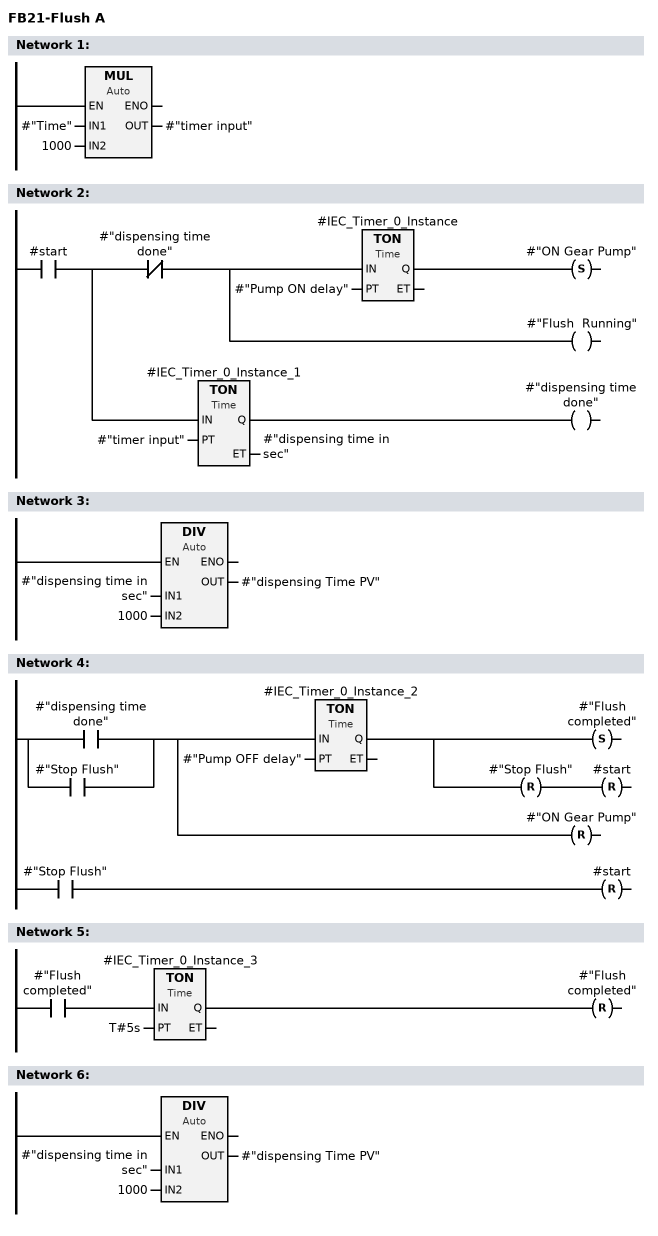
   RUNG wire#powerrail
      Mul(in1 := #"Time", in2 := 1000, out => #"timer input")
   END_RUNG
   // the same network as SCL:
   #"timer input" := #"Time" * 1000;
END_REGION

REGION Network 2
   RUNG wire#powerrail
      Contact( #start )
      wire#w1
      I_Contact( #"dispensing time done" )
      wire#w2
      { S7_Templates := "time_type := Time" } #IEC_Timer_0_Instance.TON(pt := #"Pump ON delay", et =>)
      S_Coil( #"ON Gear Pump" )
   END_RUNG
   RUNG wire#w2
      Coil( #"Flush  Running" )
   END_RUNG
   RUNG wire#w1
      { S7_Templates := "time_type := Time" } #IEC_Timer_0_Instance_1.TON(pt := #"timer input", et => #"dispensing time in sec")
      Coil( #"dispensing time done" )
   END_RUNG
   // the same network as SCL:
   #_w1 := #start AND NOT #"dispensing time done";
   #IEC_Timer_0_Instance(IN := #_w1, PT := #"Pump ON delay");   // TON
   IF #IEC_Timer_0_Instance.Q THEN #"ON Gear Pump" := TRUE; END_IF;
   #"Flush  Running" := #_w1;
   #IEC_Timer_0_Instance_1(IN := #start, PT := #"timer input", ET => #"dispensing time in sec");   // TON
   #"dispensing time done" := #IEC_Timer_0_Instance_1.Q;
END_REGION

REGION Network 3
   RUNG wire#powerrail
      Div(in1 := #"dispensing time in sec", in2 := 1000, out => #"dispensing Time PV")
   END_RUNG
   // the same network as SCL:
   #"dispensing Time PV" := #"dispensing time in sec" / 1000;
END_REGION

REGION Network 4
   RUNG wire#powerrail
      Contact( #"dispensing time done" )
      wire#w1
      { S7_Templates := "time_type := Time" } #IEC_Timer_0_Instance_2.TON(pt := #"Pump OFF delay", et =>)
      wire#w2
      S_Coil( #"Flush completed" )
   END_RUNG
   RUNG wire#powerrail
      Contact( #"Stop Flush" )
   END_RUNG wire#w1
   RUNG wire#w2
      R_Coil( #"Stop Flush" )
      R_Coil( #start )
   END_RUNG
   RUNG wire#w1
      R_Coil( #"ON Gear Pump" )
   END_RUNG
   RUNG wire#powerrail
      Contact( #"Stop Flush" )
      R_Coil( #start )
   END_RUNG
   // the same network as SCL:
   #_w1 := #"dispensing time done" OR #"Stop Flush";
   #IEC_Timer_0_Instance_2(IN := #_w1, PT := #"Pump OFF delay");   // TON
   IF #IEC_Timer_0_Instance_2.Q THEN
       #"Flush completed" := TRUE;
       #"Stop Flush" := FALSE;
       #start := FALSE;
   END_IF;
   IF #_w1 THEN #"ON Gear Pump" := FALSE; END_IF;
   IF #"Stop Flush" THEN #start := FALSE; END_IF;
END_REGION

REGION Network 5
   RUNG wire#powerrail
      Contact( #"Flush completed" )
      { S7_Templates := "time_type := Time" } #IEC_Timer_0_Instance_3.TON(pt := T#5s, et =>)
      R_Coil( #"Flush completed" )
   END_RUNG
   // the same network as SCL:
   #IEC_Timer_0_Instance_3(IN := #"Flush completed", PT := T#5s);   // TON
   IF #IEC_Timer_0_Instance_3.Q THEN #"Flush completed" := FALSE; END_IF;
END_REGION

REGION Network 6
   RUNG wire#powerrail
      Div(in1 := #"dispensing time in sec", in2 := 1000, out => #"dispensing Time PV")
   END_RUNG
   // the same network as SCL:
   #"dispensing Time PV" := #"dispensing time in sec" / 1000;
END_REGION
END_FUNCTION_BLOCK

FUNCTION "Regenaration program sequences" : Void   // FC23, LAD
{ S7_Optimized_Access := 'TRUE' }
VERSION : 0.1
// stored: AutoNumber true, IsIECCheckEnabled false, SetENOAutomatically false, UDAEnableTagReadback false
   VAR_TEMP
      temp1 : Bool;
   END_VAR
   VAR_TEMP   // added for the SCL form of the ladder/FBD networks
      _w1 : Bool;
   END_VAR
BEGIN

REGION Network 1: Function regeneration
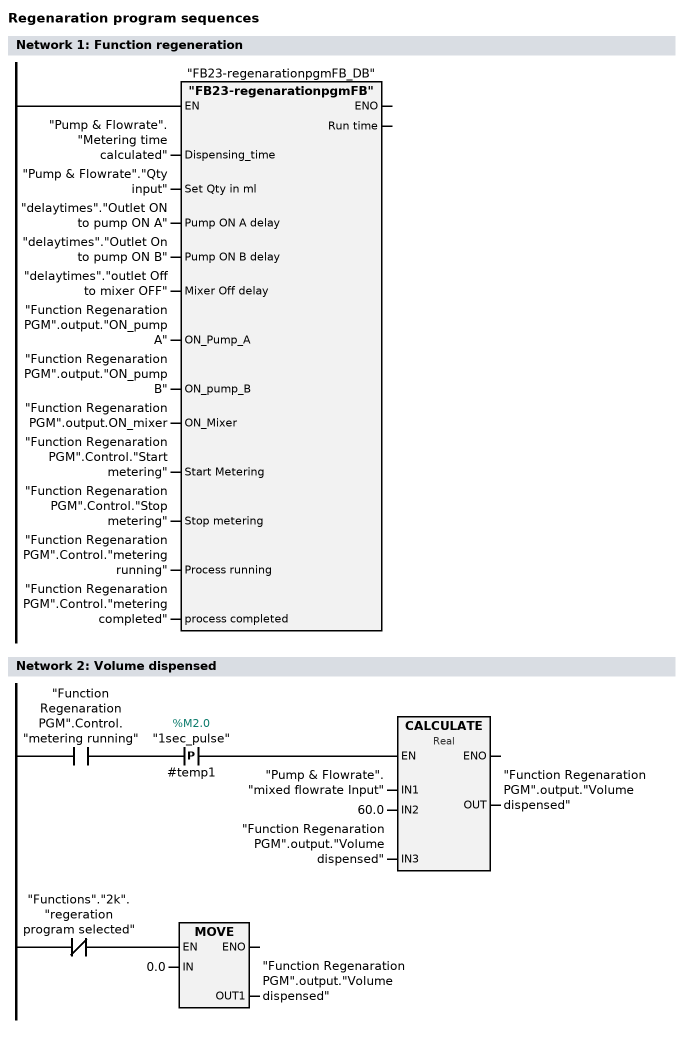
   RUNG wire#powerrail
      "FB23-regenarationpgmFB_DB"(Dispensing_time := "Pump & Flowrate"."Metering time calculated", "Set Qty in ml" := "Pump & Flowrate"."Qty input", "Pump ON A delay" := "delaytimes"."Outlet ON to pump ON A", "Pump ON B delay" := "delaytimes"."Outlet On to pump ON B", "Mixer Off delay" := "delaytimes"."outlet Off to mixer OFF", ON_Pump_A := "Function Regenaration PGM".output."ON_pump A", ON_pump_B := "Function Regenaration PGM".output."ON_pump B", ON_Mixer := "Function Regenaration PGM".output.ON_mixer, "Start Metering" := "Function Regenaration PGM".Control."Start metering", "Stop metering" := "Function Regenaration PGM".Control."Stop metering", "Process running" := "Function Regenaration PGM".Control."metering running", "process completed" := "Function Regenaration PGM".Control."metering completed", "Run time" =>)
   END_RUNG
   // the same network as SCL:
   "FB23-regenarationpgmFB_DB"(Dispensing_time := "Pump & Flowrate"."Metering time calculated",   // "FB23-regenarationpgmFB"
                           "Set Qty in ml" := "Pump & Flowrate"."Qty input",
                           "Pump ON A delay" := "delaytimes"."Outlet ON to pump ON A",
                           "Pump ON B delay" := "delaytimes"."Outlet On to pump ON B",
                           "Mixer Off delay" := "delaytimes"."outlet Off to mixer OFF",
                           ON_Pump_A := "Function Regenaration PGM".output."ON_pump A",
                           ON_pump_B := "Function Regenaration PGM".output."ON_pump B",
                           ON_Mixer := "Function Regenaration PGM".output.ON_mixer,
                           "Start Metering" := "Function Regenaration PGM".Control."Start metering",
                           "Stop metering" := "Function Regenaration PGM".Control."Stop metering",
                           "Process running" := "Function Regenaration PGM".Control."metering running",
                           "process completed" := "Function Regenaration PGM".Control."metering completed");
END_REGION

REGION Network 2: Volume dispensed
   RUNG wire#powerrail
      Contact( "Function Regenaration PGM".Control."metering running" )
      P_Contact(operand := "1sec_pulse", bit := #temp1)
      { S7_Templates := "SrcType := Real"; S7_Expression := "(IN1/IN2)+IN3" } Calculate(in1 := "Pump & Flowrate"."mixed flowrate Input", in2 := 60.0, in3 := "Function Regenaration PGM".output."Volume dispensed", out => "Function Regenaration PGM".output."Volume dispensed")
   END_RUNG
   RUNG wire#powerrail
      I_Contact( "Functions"."2k"."regeration program selected" )
      Move(in := 0.0, out1 => "Function Regenaration PGM".output."Volume dispensed")
   END_RUNG
   // the same network as SCL:
   #_w1 := "Function Regenaration PGM".Control."metering running" AND "1sec_pulse" AND NOT #temp1;   // rising edge of "1sec_pulse"
   #temp1 := "1sec_pulse";
   IF #_w1 THEN
       "Function Regenaration PGM".output."Volume dispensed" := ("Pump & Flowrate"."mixed flowrate Input"/60.0)+"Function Regenaration PGM".output."Volume dispensed";
   END_IF;
   IF NOT "Functions"."2k"."regeration program selected" THEN
       "Function Regenaration PGM".output."Volume dispensed" := 0.0;
   END_IF;
END_REGION
END_FUNCTION

FUNCTION_BLOCK "FB23-regenarationpgmFB"   // FB23, LAD
{ S7_Optimized_Access := 'TRUE' }
VERSION : 0.1
// stored: AutoNumber false, IsIECCheckEnabled false, IsRetainMemResEnabled false, MemoryReserve 100, SetENOAutomatically false, UDAEnableTagReadback false
   VAR_INPUT
      Dispensing_time : DInt;
      "Set Qty in ml" : Real;
      "Pump ON A delay" : DInt;
      "Pump ON B delay" : DInt;
      "Mixer Off delay" : DInt;
   END_VAR
   VAR_OUTPUT
      "Run time" : Int;
   END_VAR
   VAR_IN_OUT
      ON_Pump_A : Bool;
      ON_pump_B : Bool;
      ON_Mixer : Bool;
      "Start Metering" : Bool;
      "Stop metering" : Bool;
      "Process running" : Bool;
      "process completed" : Bool;
   END_VAR
   VAR
      "Total Volume dispensed" : Real;
      "metering started" : Bool;
      "metering time in msec" : DInt;
      "dispense time elapsed" : Bool;
   END_VAR
   VAR_TEMP
      Ons_temp : Bool;
   END_VAR
   VAR_TEMP   // added for the SCL form of the ladder/FBD networks
      _w1 : Bool;
   END_VAR
BEGIN

REGION Network 1
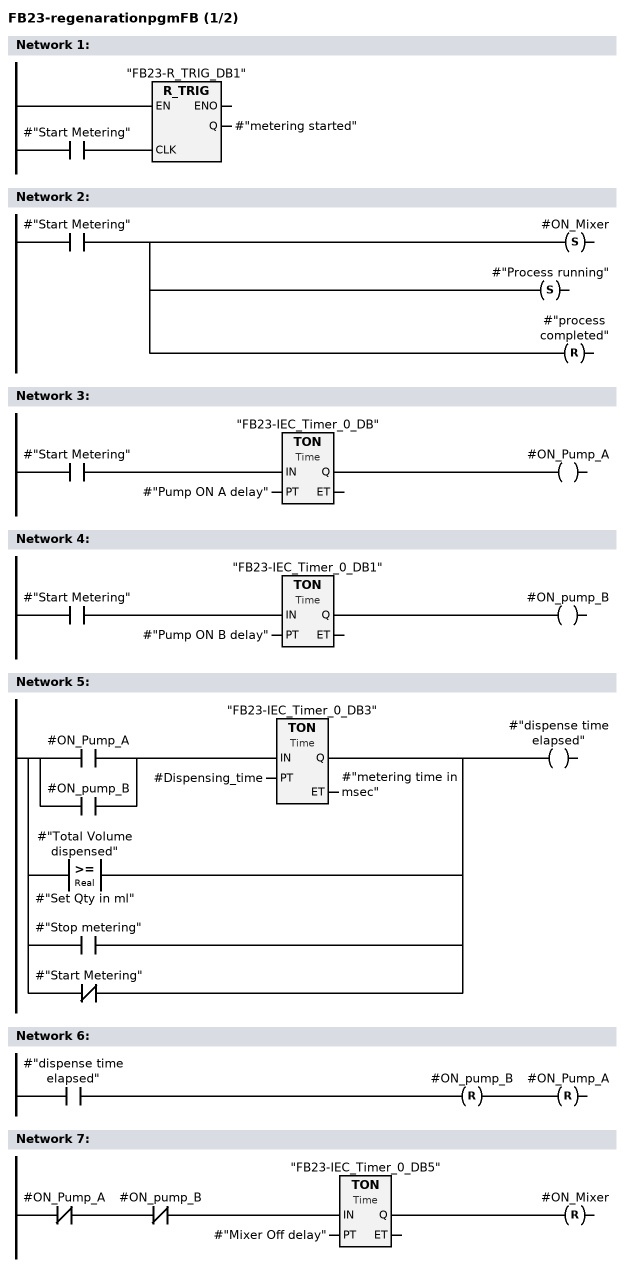
   RUNG wire#powerrail
      "FB23-R_TRIG_DB1".R_TRIG(CLK := wire#w1, Q => #"metering started")
   END_RUNG
   RUNG wire#powerrail
      Contact( #"Start Metering" )
   END_RUNG wire#w1
   // the same network as SCL:
   "FB23-R_TRIG_DB1"(CLK := #"Start Metering", Q => #"metering started");   // R_TRIG
END_REGION

REGION Network 2
   RUNG wire#powerrail
      Contact( #"Start Metering" )
      wire#w1
      S_Coil( #ON_Mixer )
   END_RUNG
   RUNG wire#w1
      S_Coil( #"Process running" )
   END_RUNG
   RUNG wire#w1
      R_Coil( #"process completed" )
   END_RUNG
   // the same network as SCL:
   IF #"Start Metering" THEN
       #ON_Mixer := TRUE;
       #"Process running" := TRUE;
       #"process completed" := FALSE;
   END_IF;
END_REGION

REGION Network 3
   RUNG wire#powerrail
      Contact( #"Start Metering" )
      { S7_Templates := "time_type := Time" } "FB23-IEC_Timer_0_DB".TON(pt := #"Pump ON A delay", et =>)
      Coil( #ON_Pump_A )
   END_RUNG
   // the same network as SCL:
   "FB23-IEC_Timer_0_DB".TON(IN := #"Start Metering", PT := #"Pump ON A delay");
   #ON_Pump_A := "FB23-IEC_Timer_0_DB".Q;
END_REGION

REGION Network 4
   RUNG wire#powerrail
      Contact( #"Start Metering" )
      { S7_Templates := "time_type := Time" } "FB23-IEC_Timer_0_DB1".TON(pt := #"Pump ON B delay", et =>)
      Coil( #ON_pump_B )
   END_RUNG
   // the same network as SCL:
   "FB23-IEC_Timer_0_DB1".TON(IN := #"Start Metering", PT := #"Pump ON B delay");
   #ON_pump_B := "FB23-IEC_Timer_0_DB1".Q;
END_REGION

REGION Network 5
   RUNG wire#powerrail
      Contact( #ON_Pump_A )
      wire#w1
      { S7_Templates := "time_type := Time" } "FB23-IEC_Timer_0_DB3".TON(pt := #Dispensing_time, et => #"metering time in msec")
      wire#w2
      Coil( #"dispense time elapsed" )
   END_RUNG
   RUNG wire#powerrail
      Contact( #ON_pump_B )
   END_RUNG wire#w1
   RUNG wire#powerrail
      { S7_Templates := "SrcType := Real" } GE_Contact(in1 := #"Total Volume dispensed", in2 := #"Set Qty in ml")
   END_RUNG wire#w2
   RUNG wire#powerrail
      Contact( #"Stop metering" )
   END_RUNG wire#w2
   RUNG wire#powerrail
      I_Contact( #"Start Metering" )
   END_RUNG wire#w2
   // the same network as SCL:
   "FB23-IEC_Timer_0_DB3".TON(IN := #ON_Pump_A OR #ON_pump_B,
                           PT := #Dispensing_time,
                           ET => #"metering time in msec");
   #"dispense time elapsed" := "FB23-IEC_Timer_0_DB3".Q OR (#"Total Volume dispensed" >= #"Set Qty in ml") OR #"Stop metering" OR NOT #"Start Metering";
END_REGION

REGION Network 6
   RUNG wire#powerrail
      Contact( #"dispense time elapsed" )
      R_Coil( #ON_pump_B )
      R_Coil( #ON_Pump_A )
   END_RUNG
   // the same network as SCL:
   IF #"dispense time elapsed" THEN
       #ON_pump_B := FALSE;
       #ON_Pump_A := FALSE;
   END_IF;
END_REGION

REGION Network 7
   RUNG wire#powerrail
      I_Contact( #ON_Pump_A )
      I_Contact( #ON_pump_B )
      { S7_Templates := "time_type := Time" } "FB23-IEC_Timer_0_DB5".TON(pt := #"Mixer Off delay", et =>)
      R_Coil( #ON_Mixer )
   END_RUNG
   // the same network as SCL:
   "FB23-IEC_Timer_0_DB5".TON(IN := NOT #ON_Pump_A AND NOT #ON_pump_B, PT := #"Mixer Off delay");
   IF "FB23-IEC_Timer_0_DB5".Q THEN #ON_Mixer := FALSE; END_IF;
END_REGION

REGION Network 8
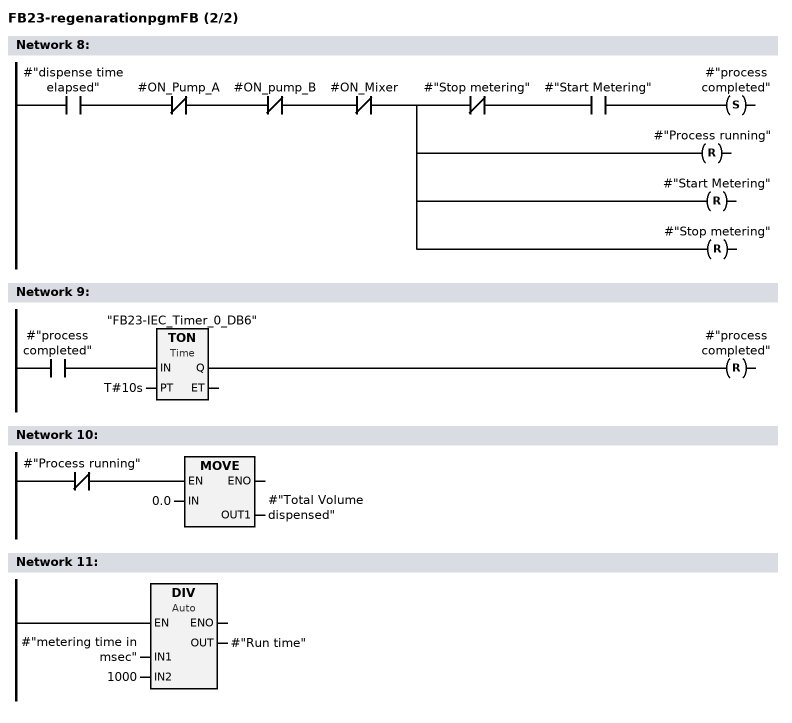
   RUNG wire#powerrail
      Contact( #"dispense time elapsed" )
      I_Contact( #ON_Pump_A )
      I_Contact( #ON_pump_B )
      I_Contact( #ON_Mixer )
      wire#w1
      I_Contact( #"Stop metering" )
      Contact( #"Start Metering" )
      S_Coil( #"process completed" )
   END_RUNG
   RUNG wire#w1
      R_Coil( #"Process running" )
   END_RUNG
   RUNG wire#w1
      R_Coil( #"Start Metering" )
   END_RUNG
   RUNG wire#w1
      R_Coil( #"Stop metering" )
   END_RUNG
   // the same network as SCL:
   #_w1 := #"dispense time elapsed" AND NOT #ON_Pump_A AND NOT #ON_pump_B AND NOT #ON_Mixer;
   IF #_w1 AND NOT #"Stop metering" AND #"Start Metering" THEN #"process completed" := TRUE; END_IF;
   IF #_w1 THEN
       #"Process running" := FALSE;
       #"Start Metering" := FALSE;
       #"Stop metering" := FALSE;
   END_IF;
END_REGION

REGION Network 9
   RUNG wire#powerrail
      Contact( #"process completed" )
      { S7_Templates := "time_type := Time" } "FB23-IEC_Timer_0_DB6".TON(pt := T#10s, et =>)
      R_Coil( #"process completed" )
   END_RUNG
   // the same network as SCL:
   "FB23-IEC_Timer_0_DB6".TON(IN := #"process completed", PT := T#10s);
   IF "FB23-IEC_Timer_0_DB6".Q THEN #"process completed" := FALSE; END_IF;
END_REGION

REGION Network 10
   RUNG wire#powerrail
      I_Contact( #"Process running" )
      Move(in := 0.0, out1 => #"Total Volume dispensed")
   END_RUNG
   // the same network as SCL:
   IF NOT #"Process running" THEN #"Total Volume dispensed" := 0.0; END_IF;
END_REGION

REGION Network 11
   RUNG wire#powerrail
      Div(in1 := #"metering time in msec", in2 := 1000, out => #"Run time")
   END_RUNG
   // the same network as SCL:
   #"Run time" := #"metering time in msec" / 1000;
END_REGION
END_FUNCTION_BLOCK

FUNCTION "Recirculation Sequences" : Void   // FC12, LAD
{ S7_Optimized_Access := 'TRUE' }
VERSION : 0.1
// stored: AutoNumber true, IsIECCheckEnabled false, SetENOAutomatically false, UDAEnableTagReadback false
   VAR_TEMP   // added for the SCL form of the ladder/FBD networks
      _w1 : Bool;
   END_VAR
BEGIN

REGION Network 1: A selection
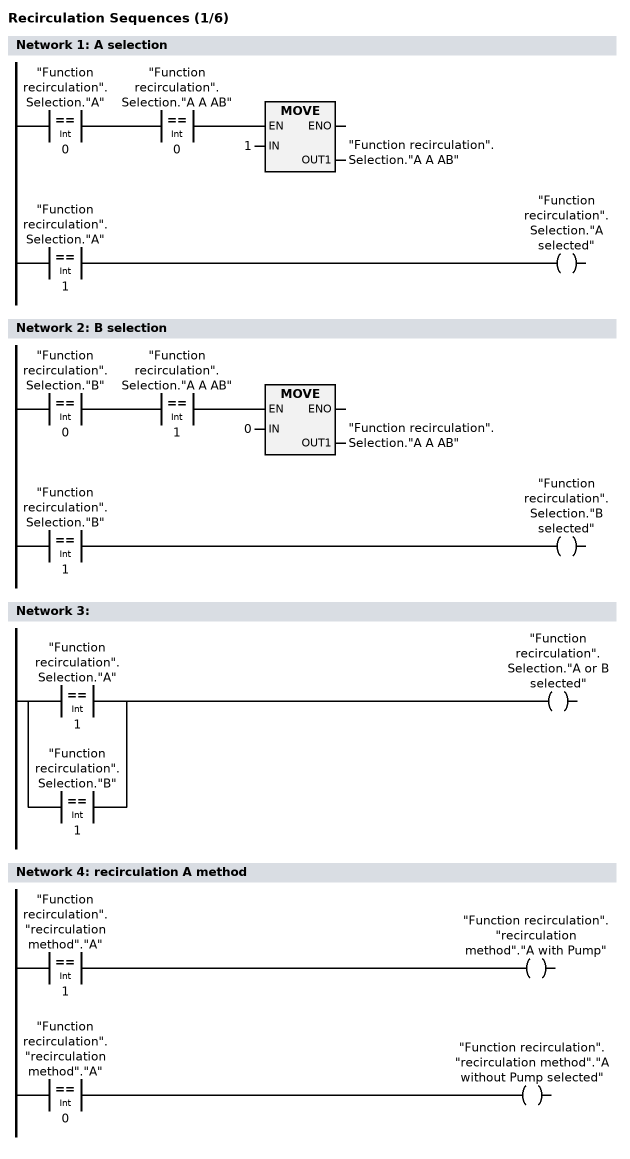
   RUNG wire#powerrail
      { S7_Templates := "SrcType := Int" } EQ_Contact(in1 := "Function recirculation".Selection."A", in2 := 0)
      { S7_Templates := "SrcType := Int" } EQ_Contact(in1 := "Function recirculation".Selection."A A AB", in2 := 0)
      Move(in := 1, out1 => "Function recirculation".Selection."A A AB")
   END_RUNG
   RUNG wire#powerrail
      { S7_Templates := "SrcType := Int" } EQ_Contact(in1 := "Function recirculation".Selection."A", in2 := 1)
      Coil( "Function recirculation".Selection."A selected" )
   END_RUNG
   // the same network as SCL:
   IF ("Function recirculation".Selection."A" = 0) AND ("Function recirculation".Selection."A A AB" = 0) THEN
       "Function recirculation".Selection."A A AB" := 1;
   END_IF;
   "Function recirculation".Selection."A selected" := "Function recirculation".Selection."A" = 1;
END_REGION

REGION Network 2: B selection
   RUNG wire#powerrail
      { S7_Templates := "SrcType := Int" } EQ_Contact(in1 := "Function recirculation".Selection."B", in2 := 0)
      { S7_Templates := "SrcType := Int" } EQ_Contact(in1 := "Function recirculation".Selection."A A AB", in2 := 1)
      Move(in := 0, out1 => "Function recirculation".Selection."A A AB")
   END_RUNG
   RUNG wire#powerrail
      { S7_Templates := "SrcType := Int" } EQ_Contact(in1 := "Function recirculation".Selection."B", in2 := 1)
      Coil( "Function recirculation".Selection."B selected" )
   END_RUNG
   // the same network as SCL:
   IF ("Function recirculation".Selection."B" = 0) AND ("Function recirculation".Selection."A A AB" = 1) THEN
       "Function recirculation".Selection."A A AB" := 0;
   END_IF;
   "Function recirculation".Selection."B selected" := "Function recirculation".Selection."B" = 1;
END_REGION

REGION Network 3
   RUNG wire#powerrail
      { S7_Templates := "SrcType := Int" } EQ_Contact(in1 := "Function recirculation".Selection."A", in2 := 1)
      wire#w1
      Coil( "Function recirculation".Selection."A or B selected" )
   END_RUNG
   RUNG wire#powerrail
      { S7_Templates := "SrcType := Int" } EQ_Contact(in1 := "Function recirculation".Selection."B", in2 := 1)
   END_RUNG wire#w1
   // the same network as SCL:
   "Function recirculation".Selection."A or B selected" := ("Function recirculation".Selection."A" = 1) OR ("Function recirculation".Selection."B" = 1);
END_REGION

REGION Network 4: recirculation A method
   RUNG wire#powerrail
      { S7_Templates := "SrcType := Int" } EQ_Contact(in1 := "Function recirculation"."recirculation method"."A", in2 := 1)
      Coil( "Function recirculation"."recirculation method"."A with Pump" )
   END_RUNG
   RUNG wire#powerrail
      { S7_Templates := "SrcType := Int" } EQ_Contact(in1 := "Function recirculation"."recirculation method"."A", in2 := 0)
      Coil( "Function recirculation"."recirculation method"."A without Pump selected" )
   END_RUNG
   // the same network as SCL:
   "Function recirculation"."recirculation method"."A with Pump" := "Function recirculation"."recirculation method"."A" = 1;
   "Function recirculation"."recirculation method"."A without Pump selected" := "Function recirculation"."recirculation method"."A" = 0;
END_REGION

REGION Network 5: recirculation B method
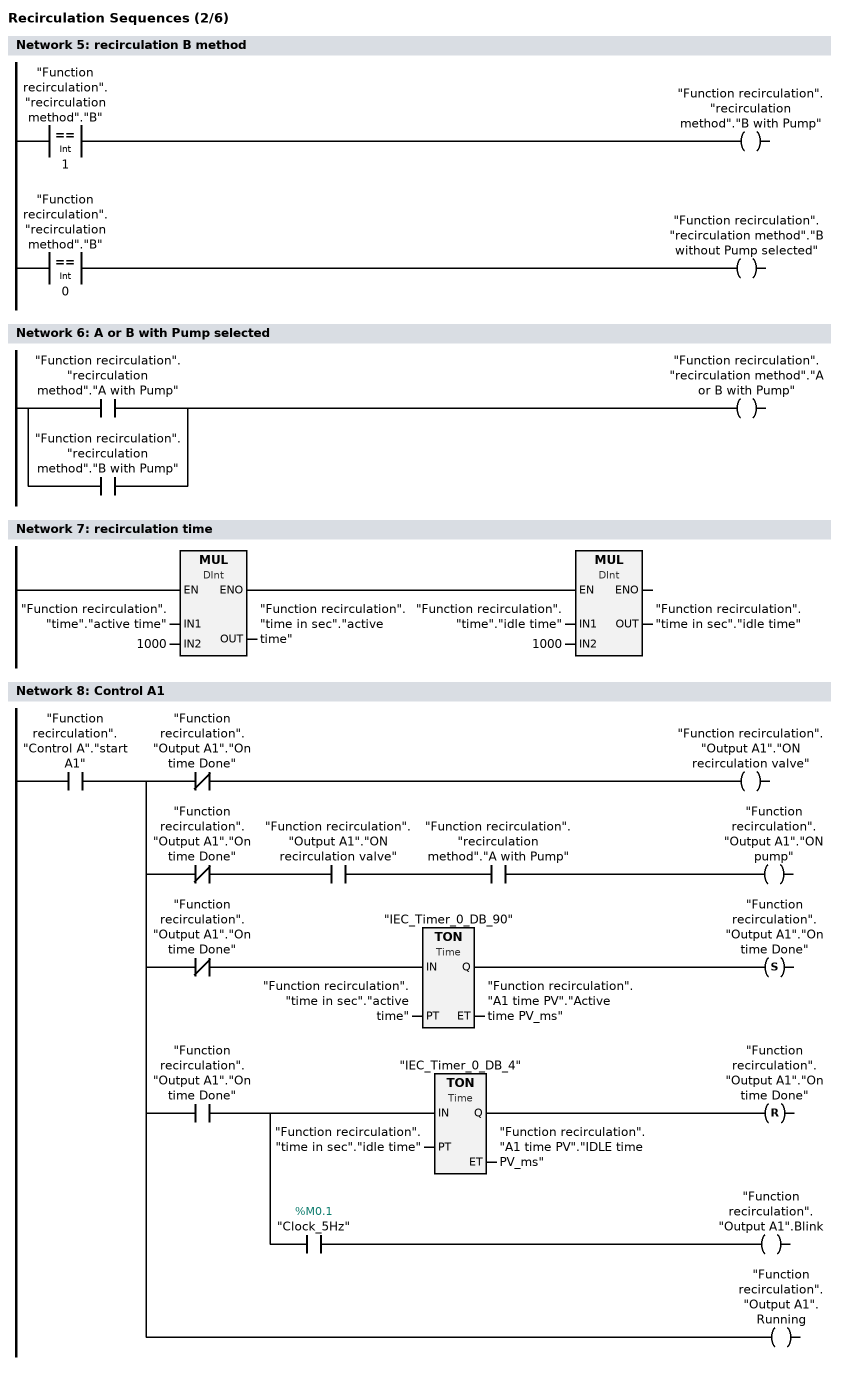
   RUNG wire#powerrail
      { S7_Templates := "SrcType := Int" } EQ_Contact(in1 := "Function recirculation"."recirculation method"."B", in2 := 1)
      Coil( "Function recirculation"."recirculation method"."B with Pump" )
   END_RUNG
   RUNG wire#powerrail
      { S7_Templates := "SrcType := Int" } EQ_Contact(in1 := "Function recirculation"."recirculation method"."B", in2 := 0)
      Coil( "Function recirculation"."recirculation method"."B without Pump selected" )
   END_RUNG
   // the same network as SCL:
   "Function recirculation"."recirculation method"."B with Pump" := "Function recirculation"."recirculation method"."B" = 1;
   "Function recirculation"."recirculation method"."B without Pump selected" := "Function recirculation"."recirculation method"."B" = 0;
END_REGION

REGION Network 6: A or B with Pump selected
   RUNG wire#powerrail
      Contact( "Function recirculation"."recirculation method"."A with Pump" )
      wire#w1
      Coil( "Function recirculation"."recirculation method"."A or B with Pump" )
   END_RUNG
   RUNG wire#powerrail
      Contact( "Function recirculation"."recirculation method"."B with Pump" )
   END_RUNG wire#w1
   // the same network as SCL:
   "Function recirculation"."recirculation method"."A or B with Pump" := "Function recirculation"."recirculation method"."A with Pump" OR "Function recirculation"."recirculation method"."B with Pump";
END_REGION

REGION Network 7: recirculation time
   RUNG wire#powerrail
      { S7_Templates := "SrcType := DInt" } Mul(in1 := "Function recirculation"."time"."active time", in2 := 1000, out => "Function recirculation"."time in sec"."active time")
      { S7_Templates := "SrcType := DInt" } Mul(in1 := "Function recirculation"."time"."idle time", in2 := 1000, out => "Function recirculation"."time in sec"."idle time")
   END_RUNG
   // the same network as SCL:
   "Function recirculation"."time in sec"."active time" := "Function recirculation"."time"."active time" * 1000;
   "Function recirculation"."time in sec"."idle time" := "Function recirculation"."time"."idle time" * 1000;
END_REGION

REGION Network 8: Control A1
   RUNG wire#powerrail
      Contact( "Function recirculation"."Control A"."start A1" )
      wire#w1
      I_Contact( "Function recirculation"."Output A1"."On time Done" )
      Coil( "Function recirculation"."Output A1"."ON recirculation valve" )
   END_RUNG
   RUNG wire#w1
      I_Contact( "Function recirculation"."Output A1"."On time Done" )
      Contact( "Function recirculation"."Output A1"."ON recirculation valve" )
      Contact( "Function recirculation"."recirculation method"."A with Pump" )
      Coil( "Function recirculation"."Output A1"."ON pump" )
   END_RUNG
   RUNG wire#w1
      I_Contact( "Function recirculation"."Output A1"."On time Done" )
      { S7_Templates := "time_type := Time" } "IEC_Timer_0_DB_90".TON(pt := "Function recirculation"."time in sec"."active time", et => "Function recirculation"."A1 time PV"."Active time PV_ms")
      S_Coil( "Function recirculation"."Output A1"."On time Done" )
   END_RUNG
   RUNG wire#w1
      Contact( "Function recirculation"."Output A1"."On time Done" )
      wire#w2
      { S7_Templates := "time_type := Time" } "IEC_Timer_0_DB_4".TON(pt := "Function recirculation"."time in sec"."idle time", et => "Function recirculation"."A1 time PV"."IDLE time PV_ms")
      R_Coil( "Function recirculation"."Output A1"."On time Done" )
   END_RUNG
   RUNG wire#w2
      Contact( "Clock_5Hz" )
      Coil( "Function recirculation"."Output A1".Blink )
   END_RUNG
   RUNG wire#w1
      Coil( "Function recirculation"."Output A1".Running )
   END_RUNG
   // the same network as SCL:
   "Function recirculation"."Output A1"."ON recirculation valve" := "Function recirculation"."Control A"."start A1" AND NOT "Function recirculation"."Output A1"."On time Done";
   "Function recirculation"."Output A1"."ON pump" := "Function recirculation"."Control A"."start A1" AND NOT "Function recirculation"."Output A1"."On time Done" AND "Function recirculation"."Output A1"."ON recirculation valve" AND "Function recirculation"."recirculation method"."A with Pump";
   "IEC_Timer_0_DB_90".TON(IN := "Function recirculation"."Control A"."start A1" AND NOT "Function recirculation"."Output A1"."On time Done",
                           PT := "Function recirculation"."time in sec"."active time",
                           ET => "Function recirculation"."A1 time PV"."Active time PV_ms");
   IF "IEC_Timer_0_DB_90".Q THEN "Function recirculation"."Output A1"."On time Done" := TRUE; END_IF;
   #_w1 := "Function recirculation"."Control A"."start A1" AND "Function recirculation"."Output A1"."On time Done";
   "IEC_Timer_0_DB_4".TON(IN := #_w1,
                          PT := "Function recirculation"."time in sec"."idle time",
                          ET => "Function recirculation"."A1 time PV"."IDLE time PV_ms");
   IF "IEC_Timer_0_DB_4".Q THEN "Function recirculation"."Output A1"."On time Done" := FALSE; END_IF;
   "Function recirculation"."Output A1".Blink := #_w1 AND "Clock_5Hz";
   "Function recirculation"."Output A1".Running := "Function recirculation"."Control A"."start A1";
END_REGION

REGION Network 9: Control A2
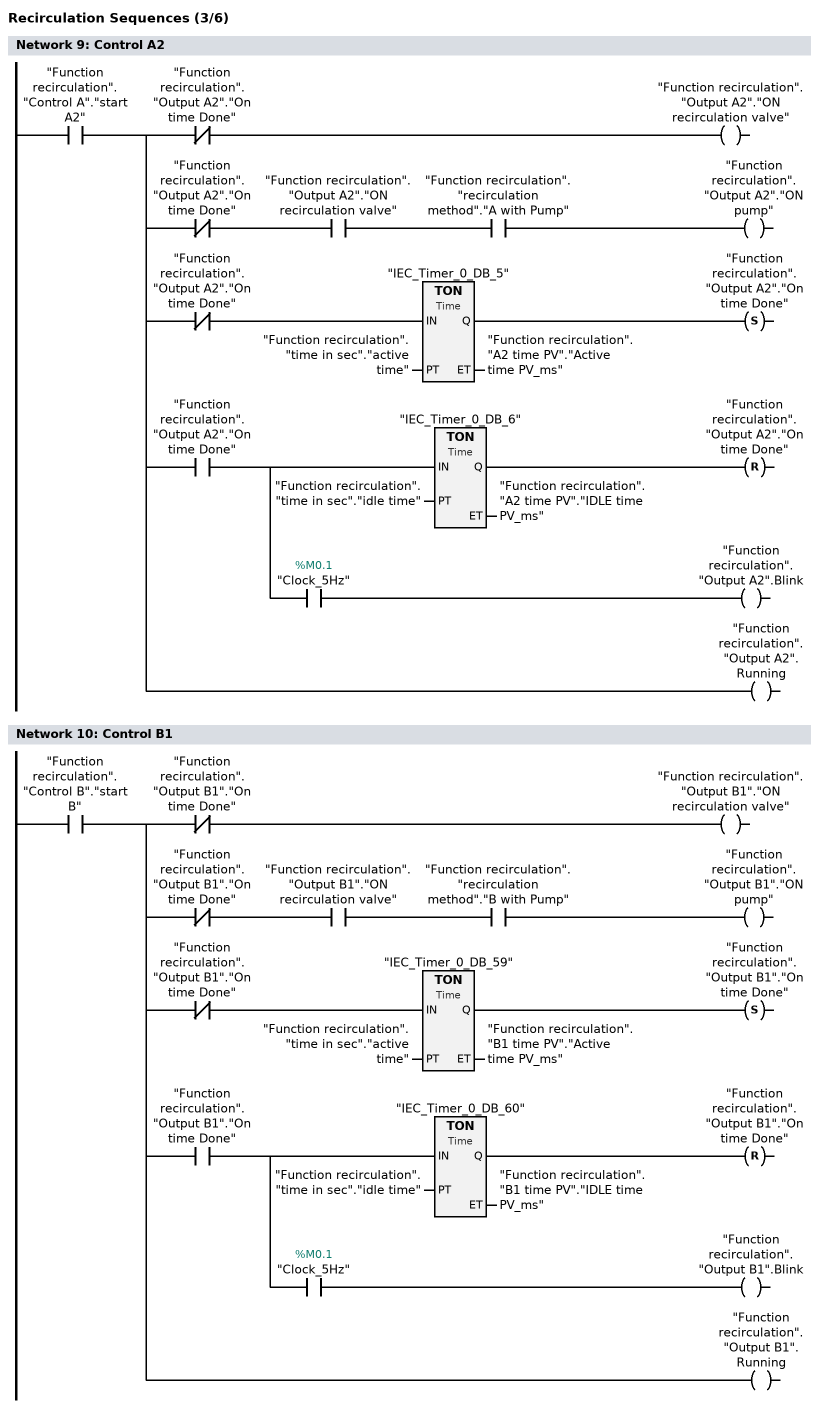
   RUNG wire#powerrail
      Contact( "Function recirculation"."Control A"."start A2" )
      wire#w1
      I_Contact( "Function recirculation"."Output A2"."On time Done" )
      Coil( "Function recirculation"."Output A2"."ON recirculation valve" )
   END_RUNG
   RUNG wire#w1
      I_Contact( "Function recirculation"."Output A2"."On time Done" )
      Contact( "Function recirculation"."Output A2"."ON recirculation valve" )
      Contact( "Function recirculation"."recirculation method"."A with Pump" )
      Coil( "Function recirculation"."Output A2"."ON pump" )
   END_RUNG
   RUNG wire#w1
      I_Contact( "Function recirculation"."Output A2"."On time Done" )
      { S7_Templates := "time_type := Time" } "IEC_Timer_0_DB_5".TON(pt := "Function recirculation"."time in sec"."active time", et => "Function recirculation"."A2 time PV"."Active time PV_ms")
      S_Coil( "Function recirculation"."Output A2"."On time Done" )
   END_RUNG
   RUNG wire#w1
      Contact( "Function recirculation"."Output A2"."On time Done" )
      wire#w2
      { S7_Templates := "time_type := Time" } "IEC_Timer_0_DB_6".TON(pt := "Function recirculation"."time in sec"."idle time", et => "Function recirculation"."A2 time PV"."IDLE time PV_ms")
      R_Coil( "Function recirculation"."Output A2"."On time Done" )
   END_RUNG
   RUNG wire#w2
      Contact( "Clock_5Hz" )
      Coil( "Function recirculation"."Output A2".Blink )
   END_RUNG
   RUNG wire#w1
      Coil( "Function recirculation"."Output A2".Running )
   END_RUNG
   // the same network as SCL:
   "Function recirculation"."Output A2"."ON recirculation valve" := "Function recirculation"."Control A"."start A2" AND NOT "Function recirculation"."Output A2"."On time Done";
   "Function recirculation"."Output A2"."ON pump" := "Function recirculation"."Control A"."start A2" AND NOT "Function recirculation"."Output A2"."On time Done" AND "Function recirculation"."Output A2"."ON recirculation valve" AND "Function recirculation"."recirculation method"."A with Pump";
   "IEC_Timer_0_DB_5".TON(IN := "Function recirculation"."Control A"."start A2" AND NOT "Function recirculation"."Output A2"."On time Done",
                          PT := "Function recirculation"."time in sec"."active time",
                          ET => "Function recirculation"."A2 time PV"."Active time PV_ms");
   IF "IEC_Timer_0_DB_5".Q THEN "Function recirculation"."Output A2"."On time Done" := TRUE; END_IF;
   #_w1 := "Function recirculation"."Control A"."start A2" AND "Function recirculation"."Output A2"."On time Done";
   "IEC_Timer_0_DB_6".TON(IN := #_w1,
                          PT := "Function recirculation"."time in sec"."idle time",
                          ET => "Function recirculation"."A2 time PV"."IDLE time PV_ms");
   IF "IEC_Timer_0_DB_6".Q THEN "Function recirculation"."Output A2"."On time Done" := FALSE; END_IF;
   "Function recirculation"."Output A2".Blink := #_w1 AND "Clock_5Hz";
   "Function recirculation"."Output A2".Running := "Function recirculation"."Control A"."start A2";
END_REGION

REGION Network 10: Control B1
   RUNG wire#powerrail
      Contact( "Function recirculation"."Control B"."start B" )
      wire#w1
      I_Contact( "Function recirculation"."Output B1"."On time Done" )
      Coil( "Function recirculation"."Output B1"."ON recirculation valve" )
   END_RUNG
   RUNG wire#w1
      I_Contact( "Function recirculation"."Output B1"."On time Done" )
      Contact( "Function recirculation"."Output B1"."ON recirculation valve" )
      Contact( "Function recirculation"."recirculation method"."B with Pump" )
      Coil( "Function recirculation"."Output B1"."ON pump" )
   END_RUNG
   RUNG wire#w1
      I_Contact( "Function recirculation"."Output B1"."On time Done" )
      { S7_Templates := "time_type := Time" } "IEC_Timer_0_DB_59".TON(pt := "Function recirculation"."time in sec"."active time", et => "Function recirculation"."B1 time PV"."Active time PV_ms")
      S_Coil( "Function recirculation"."Output B1"."On time Done" )
   END_RUNG
   RUNG wire#w1
      Contact( "Function recirculation"."Output B1"."On time Done" )
      wire#w2
      { S7_Templates := "time_type := Time" } "IEC_Timer_0_DB_60".TON(pt := "Function recirculation"."time in sec"."idle time", et => "Function recirculation"."B1 time PV"."IDLE time PV_ms")
      R_Coil( "Function recirculation"."Output B1"."On time Done" )
   END_RUNG
   RUNG wire#w2
      Contact( "Clock_5Hz" )
      Coil( "Function recirculation"."Output B1".Blink )
   END_RUNG
   RUNG wire#w1
      Coil( "Function recirculation"."Output B1".Running )
   END_RUNG
   // the same network as SCL:
   "Function recirculation"."Output B1"."ON recirculation valve" := "Function recirculation"."Control B"."start B" AND NOT "Function recirculation"."Output B1"."On time Done";
   "Function recirculation"."Output B1"."ON pump" := "Function recirculation"."Control B"."start B" AND NOT "Function recirculation"."Output B1"."On time Done" AND "Function recirculation"."Output B1"."ON recirculation valve" AND "Function recirculation"."recirculation method"."B with Pump";
   "IEC_Timer_0_DB_59".TON(IN := "Function recirculation"."Control B"."start B" AND NOT "Function recirculation"."Output B1"."On time Done",
                           PT := "Function recirculation"."time in sec"."active time",
                           ET => "Function recirculation"."B1 time PV"."Active time PV_ms");
   IF "IEC_Timer_0_DB_59".Q THEN "Function recirculation"."Output B1"."On time Done" := TRUE; END_IF;
   #_w1 := "Function recirculation"."Control B"."start B" AND "Function recirculation"."Output B1"."On time Done";
   "IEC_Timer_0_DB_60".TON(IN := #_w1,
                           PT := "Function recirculation"."time in sec"."idle time",
                           ET => "Function recirculation"."B1 time PV"."IDLE time PV_ms");
   IF "IEC_Timer_0_DB_60".Q THEN "Function recirculation"."Output B1"."On time Done" := FALSE; END_IF;
   "Function recirculation"."Output B1".Blink := #_w1 AND "Clock_5Hz";
   "Function recirculation"."Output B1".Running := "Function recirculation"."Control B"."start B";
END_REGION

REGION Network 11: Recirculation A Active time PV
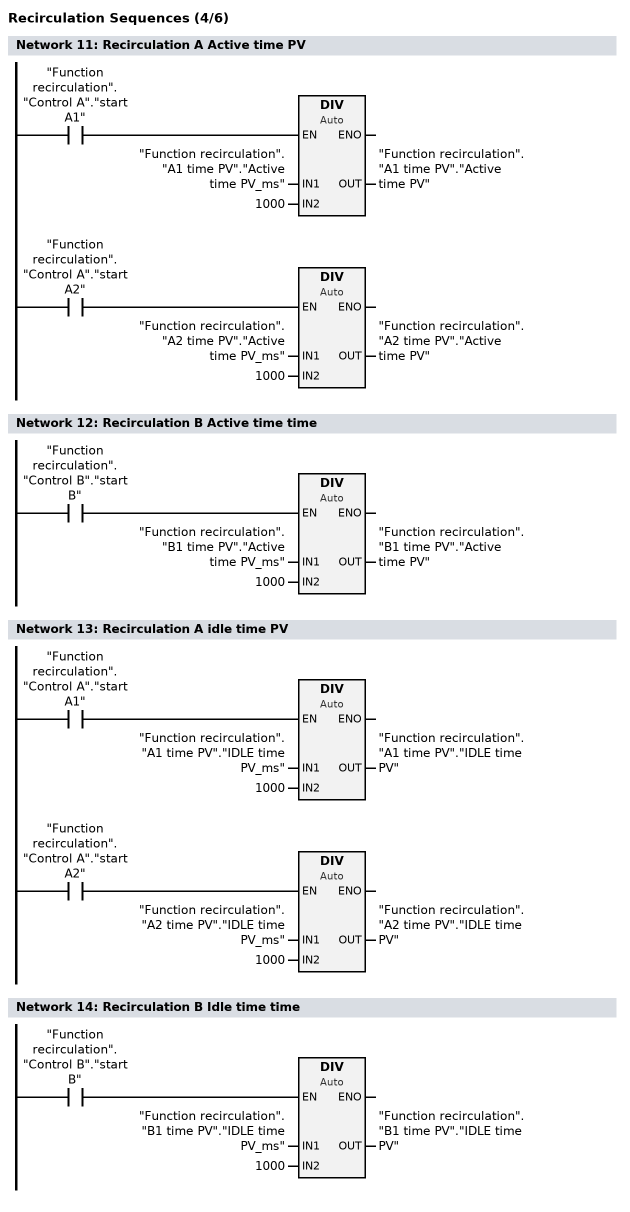
   RUNG wire#powerrail
      Contact( "Function recirculation"."Control A"."start A1" )
      Div(in1 := "Function recirculation"."A1 time PV"."Active time PV_ms", in2 := 1000, out => "Function recirculation"."A1 time PV"."Active time PV")
   END_RUNG
   RUNG wire#powerrail
      Contact( "Function recirculation"."Control A"."start A2" )
      Div(in1 := "Function recirculation"."A2 time PV"."Active time PV_ms", in2 := 1000, out => "Function recirculation"."A2 time PV"."Active time PV")
   END_RUNG
   // the same network as SCL:
   IF "Function recirculation"."Control A"."start A1" THEN
       "Function recirculation"."A1 time PV"."Active time PV" := "Function recirculation"."A1 time PV"."Active time PV_ms" / 1000;
   END_IF;
   IF "Function recirculation"."Control A"."start A2" THEN
       "Function recirculation"."A2 time PV"."Active time PV" := "Function recirculation"."A2 time PV"."Active time PV_ms" / 1000;
   END_IF;
END_REGION

REGION Network 12: Recirculation B Active time time
   RUNG wire#powerrail
      Contact( "Function recirculation"."Control B"."start B" )
      Div(in1 := "Function recirculation"."B1 time PV"."Active time PV_ms", in2 := 1000, out => "Function recirculation"."B1 time PV"."Active time PV")
   END_RUNG
   // the same network as SCL:
   IF "Function recirculation"."Control B"."start B" THEN
       "Function recirculation"."B1 time PV"."Active time PV" := "Function recirculation"."B1 time PV"."Active time PV_ms" / 1000;
   END_IF;
END_REGION

REGION Network 13: Recirculation A idle time PV
   RUNG wire#powerrail
      Contact( "Function recirculation"."Control A"."start A1" )
      Div(in1 := "Function recirculation"."A1 time PV"."IDLE time PV_ms", in2 := 1000, out => "Function recirculation"."A1 time PV"."IDLE time PV")
   END_RUNG
   RUNG wire#powerrail
      Contact( "Function recirculation"."Control A"."start A2" )
      Div(in1 := "Function recirculation"."A2 time PV"."IDLE time PV_ms", in2 := 1000, out => "Function recirculation"."A2 time PV"."IDLE time PV")
   END_RUNG
   // the same network as SCL:
   IF "Function recirculation"."Control A"."start A1" THEN
       "Function recirculation"."A1 time PV"."IDLE time PV" := "Function recirculation"."A1 time PV"."IDLE time PV_ms" / 1000;
   END_IF;
   IF "Function recirculation"."Control A"."start A2" THEN
       "Function recirculation"."A2 time PV"."IDLE time PV" := "Function recirculation"."A2 time PV"."IDLE time PV_ms" / 1000;
   END_IF;
END_REGION

REGION Network 14: Recirculation B Idle time time
   RUNG wire#powerrail
      Contact( "Function recirculation"."Control B"."start B" )
      Div(in1 := "Function recirculation"."B1 time PV"."IDLE time PV_ms", in2 := 1000, out => "Function recirculation"."B1 time PV"."IDLE time PV")
   END_RUNG
   // the same network as SCL:
   IF "Function recirculation"."Control B"."start B" THEN
       "Function recirculation"."B1 time PV"."IDLE time PV" := "Function recirculation"."B1 time PV"."IDLE time PV_ms" / 1000;
   END_IF;
END_REGION

REGION Network 15: A1 Active time to HMI
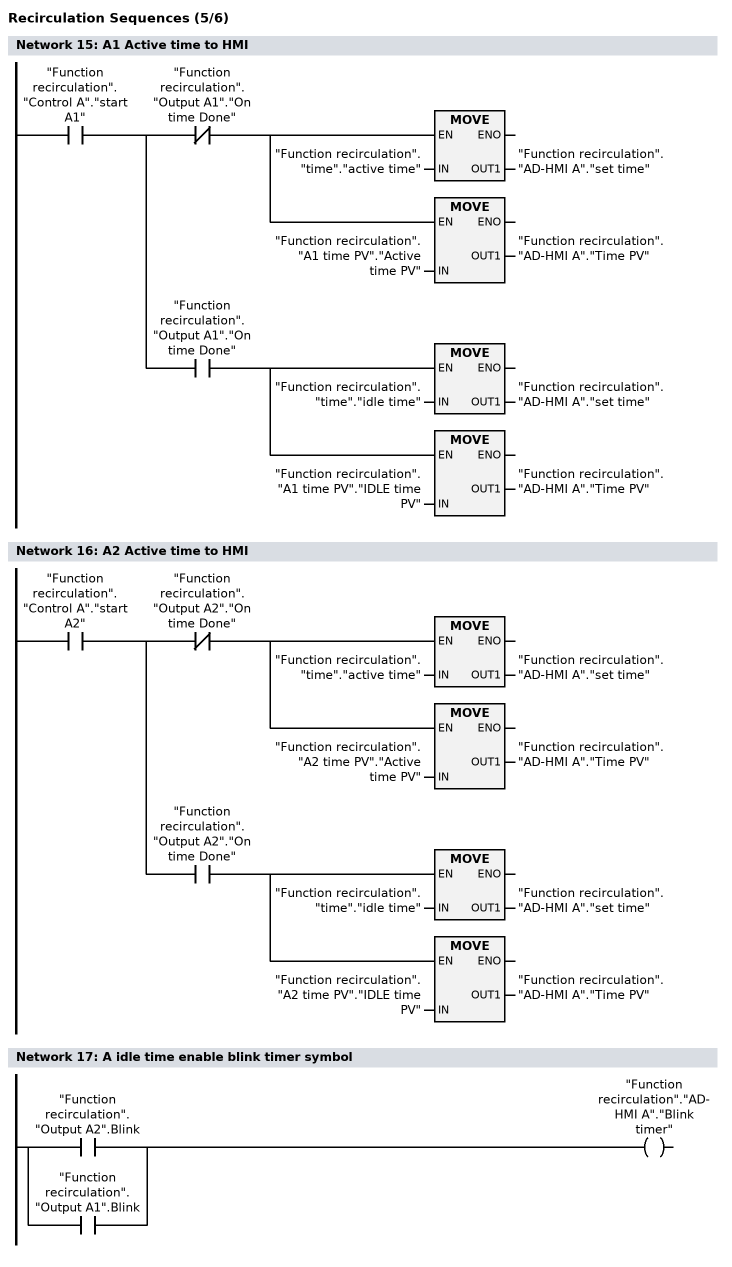
   RUNG wire#powerrail
      Contact( "Function recirculation"."Control A"."start A1" )
      wire#w1
      I_Contact( "Function recirculation"."Output A1"."On time Done" )
      wire#w2
      Move(in := "Function recirculation"."time"."active time", out1 => "Function recirculation"."AD-HMI A"."set time")
   END_RUNG
   RUNG wire#w2
      Move(in := "Function recirculation"."A1 time PV"."Active time PV", out1 => "Function recirculation"."AD-HMI A"."Time PV")
   END_RUNG
   RUNG wire#w1
      Contact( "Function recirculation"."Output A1"."On time Done" )
      wire#w3
      Move(in := "Function recirculation"."time"."idle time", out1 => "Function recirculation"."AD-HMI A"."set time")
   END_RUNG
   RUNG wire#w3
      Move(in := "Function recirculation"."A1 time PV"."IDLE time PV", out1 => "Function recirculation"."AD-HMI A"."Time PV")
   END_RUNG
   // the same network as SCL:
   IF "Function recirculation"."Control A"."start A1" AND NOT "Function recirculation"."Output A1"."On time Done" THEN
       "Function recirculation"."AD-HMI A"."set time" := "Function recirculation"."time"."active time";
       "Function recirculation"."AD-HMI A"."Time PV" := "Function recirculation"."A1 time PV"."Active time PV";
   END_IF;
   IF "Function recirculation"."Control A"."start A1" AND "Function recirculation"."Output A1"."On time Done" THEN
       "Function recirculation"."AD-HMI A"."set time" := "Function recirculation"."time"."idle time";
       "Function recirculation"."AD-HMI A"."Time PV" := "Function recirculation"."A1 time PV"."IDLE time PV";
   END_IF;
END_REGION

REGION Network 16: A2 Active time to HMI
   RUNG wire#powerrail
      Contact( "Function recirculation"."Control A"."start A2" )
      wire#w1
      I_Contact( "Function recirculation"."Output A2"."On time Done" )
      wire#w2
      Move(in := "Function recirculation"."time"."active time", out1 => "Function recirculation"."AD-HMI A"."set time")
   END_RUNG
   RUNG wire#w2
      Move(in := "Function recirculation"."A2 time PV"."Active time PV", out1 => "Function recirculation"."AD-HMI A"."Time PV")
   END_RUNG
   RUNG wire#w1
      Contact( "Function recirculation"."Output A2"."On time Done" )
      wire#w3
      Move(in := "Function recirculation"."time"."idle time", out1 => "Function recirculation"."AD-HMI A"."set time")
   END_RUNG
   RUNG wire#w3
      Move(in := "Function recirculation"."A2 time PV"."IDLE time PV", out1 => "Function recirculation"."AD-HMI A"."Time PV")
   END_RUNG
   // the same network as SCL:
   IF "Function recirculation"."Control A"."start A2" AND NOT "Function recirculation"."Output A2"."On time Done" THEN
       "Function recirculation"."AD-HMI A"."set time" := "Function recirculation"."time"."active time";
       "Function recirculation"."AD-HMI A"."Time PV" := "Function recirculation"."A2 time PV"."Active time PV";
   END_IF;
   IF "Function recirculation"."Control A"."start A2" AND "Function recirculation"."Output A2"."On time Done" THEN
       "Function recirculation"."AD-HMI A"."set time" := "Function recirculation"."time"."idle time";
       "Function recirculation"."AD-HMI A"."Time PV" := "Function recirculation"."A2 time PV"."IDLE time PV";
   END_IF;
END_REGION

REGION Network 17: A idle time enable blink timer symbol
   RUNG wire#powerrail
      Contact( "Function recirculation"."Output A2".Blink )
      wire#w1
      Coil( "Function recirculation"."AD-HMI A"."Blink timer" )
   END_RUNG
   RUNG wire#powerrail
      Contact( "Function recirculation"."Output A1".Blink )
   END_RUNG wire#w1
   // the same network as SCL:
   "Function recirculation"."AD-HMI A"."Blink timer" := "Function recirculation"."Output A2".Blink OR "Function recirculation"."Output A1".Blink;
END_REGION

REGION Network 18: B Active time to HMI
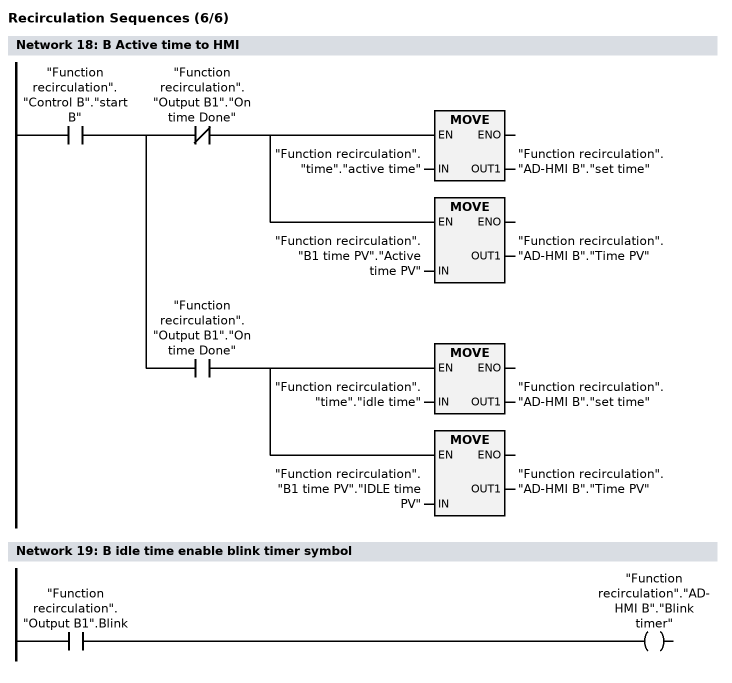
   RUNG wire#powerrail
      Contact( "Function recirculation"."Control B"."start B" )
      wire#w1
      I_Contact( "Function recirculation"."Output B1"."On time Done" )
      wire#w2
      Move(in := "Function recirculation"."time"."active time", out1 => "Function recirculation"."AD-HMI B"."set time")
   END_RUNG
   RUNG wire#w2
      Move(in := "Function recirculation"."B1 time PV"."Active time PV", out1 => "Function recirculation"."AD-HMI B"."Time PV")
   END_RUNG
   RUNG wire#w1
      Contact( "Function recirculation"."Output B1"."On time Done" )
      wire#w3
      Move(in := "Function recirculation"."time"."idle time", out1 => "Function recirculation"."AD-HMI B"."set time")
   END_RUNG
   RUNG wire#w3
      Move(in := "Function recirculation"."B1 time PV"."IDLE time PV", out1 => "Function recirculation"."AD-HMI B"."Time PV")
   END_RUNG
   // the same network as SCL:
   IF "Function recirculation"."Control B"."start B" AND NOT "Function recirculation"."Output B1"."On time Done" THEN
       "Function recirculation"."AD-HMI B"."set time" := "Function recirculation"."time"."active time";
       "Function recirculation"."AD-HMI B"."Time PV" := "Function recirculation"."B1 time PV"."Active time PV";
   END_IF;
   IF "Function recirculation"."Control B"."start B" AND "Function recirculation"."Output B1"."On time Done" THEN
       "Function recirculation"."AD-HMI B"."set time" := "Function recirculation"."time"."idle time";
       "Function recirculation"."AD-HMI B"."Time PV" := "Function recirculation"."B1 time PV"."IDLE time PV";
   END_IF;
END_REGION

REGION Network 19: B idle time enable blink timer symbol
   RUNG wire#powerrail
      Contact( "Function recirculation"."Output B1".Blink )
      Coil( "Function recirculation"."AD-HMI B"."Blink timer" )
   END_RUNG
   // the same network as SCL:
   "Function recirculation"."AD-HMI B"."Blink timer" := "Function recirculation"."Output B1".Blink;
END_REGION
END_FUNCTION

FUNCTION "recipe" : Void   // FC19, LAD
{ S7_Optimized_Access := 'TRUE' }
VERSION : 0.1
// stored: AutoNumber true, IsIECCheckEnabled false, SetENOAutomatically false, UDAEnableTagReadback false
BEGIN

REGION Network 1: program No from site
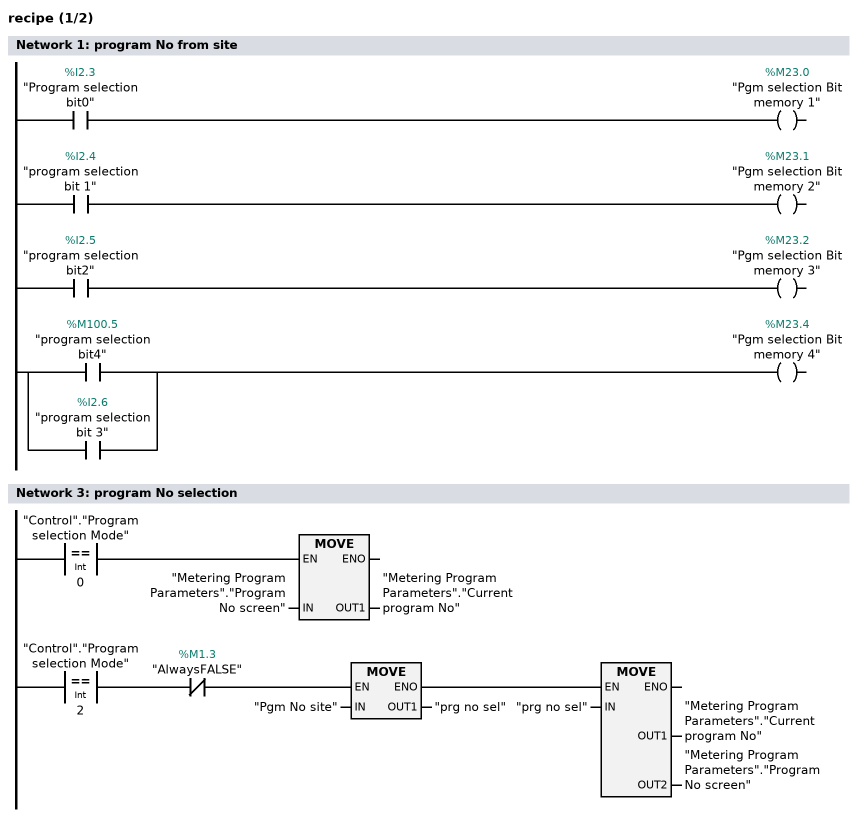
   RUNG wire#powerrail
      Contact( "Program selection bit0" )
      Coil( "Pgm selection Bit memory 1" )
   END_RUNG
   RUNG wire#powerrail
      Contact( "program selection bit 1" )
      Coil( "Pgm selection Bit memory 2" )
   END_RUNG
   RUNG wire#powerrail
      Contact( "program selection bit2" )
      Coil( "Pgm selection Bit memory 3" )
   END_RUNG
   RUNG wire#powerrail
      Contact( "program selection bit4" )
      wire#w1
      Coil( "Pgm selection Bit memory 4" )
   END_RUNG
   RUNG wire#powerrail
      Contact( "program selection bit 3" )
   END_RUNG wire#w1
   // the same network as SCL:
   "Pgm selection Bit memory 1" := "Program selection bit0";
   "Pgm selection Bit memory 2" := "program selection bit 1";
   "Pgm selection Bit memory 3" := "program selection bit2";
   "Pgm selection Bit memory 4" := "program selection bit4" OR "program selection bit 3";
END_REGION

REGION Network 2 (SCL)
   IF "Control"."Program selection Mode" = 1 THEN
     IF "Pgm selection Bit memory 1" THEN
       "Metering Program Parameters"."Receipe Program No" := 1;
     ELSIF "Pgm selection Bit memory 2" THEN
       "Metering Program Parameters"."Receipe Program No" := 2;
     ELSIF "Pgm selection Bit memory 3" THEN
       "Metering Program Parameters"."Receipe Program No" := 3;
     ELSIF "Pgm selection Bit memory 4" THEN
       "Metering Program Parameters"."Receipe Program No" := 4;
     ELSE
       "Metering Program Parameters"."Receipe Program No" := 0;
     END_IF;
   END_IF;
END_REGION

REGION Network 3: program No selection
   RUNG wire#powerrail
      { S7_Templates := "SrcType := Int" } EQ_Contact(in1 := "Control"."Program selection Mode", in2 := 0)
      Move(in := "Metering Program Parameters"."Program No screen", out1 => "Metering Program Parameters"."Current program No")
   END_RUNG
   RUNG wire#powerrail
      { S7_Templates := "SrcType := Int" } EQ_Contact(in1 := "Control"."Program selection Mode", in2 := 2)
      I_Contact( "AlwaysFALSE" )
      Move(in := "Pgm No site", out1 => "prg no sel")
      Move(in := "prg no sel", out1 => "Metering Program Parameters"."Current program No", out2 => "Metering Program Parameters"."Program No screen")
   END_RUNG
   // the same network as SCL:
   IF "Control"."Program selection Mode" = 0 THEN
       "Metering Program Parameters"."Current program No" := "Metering Program Parameters"."Program No screen";
   END_IF;
   IF ("Control"."Program selection Mode" = 2) AND NOT "AlwaysFALSE" THEN
       "prg no sel" := "Pgm No site";
       "Metering Program Parameters"."Current program No" := "prg no sel";
       "Metering Program Parameters"."Program No screen" := "prg no sel";
   END_IF;
END_REGION

REGION Network 4: Current flowrate qty and flowrate adjustment
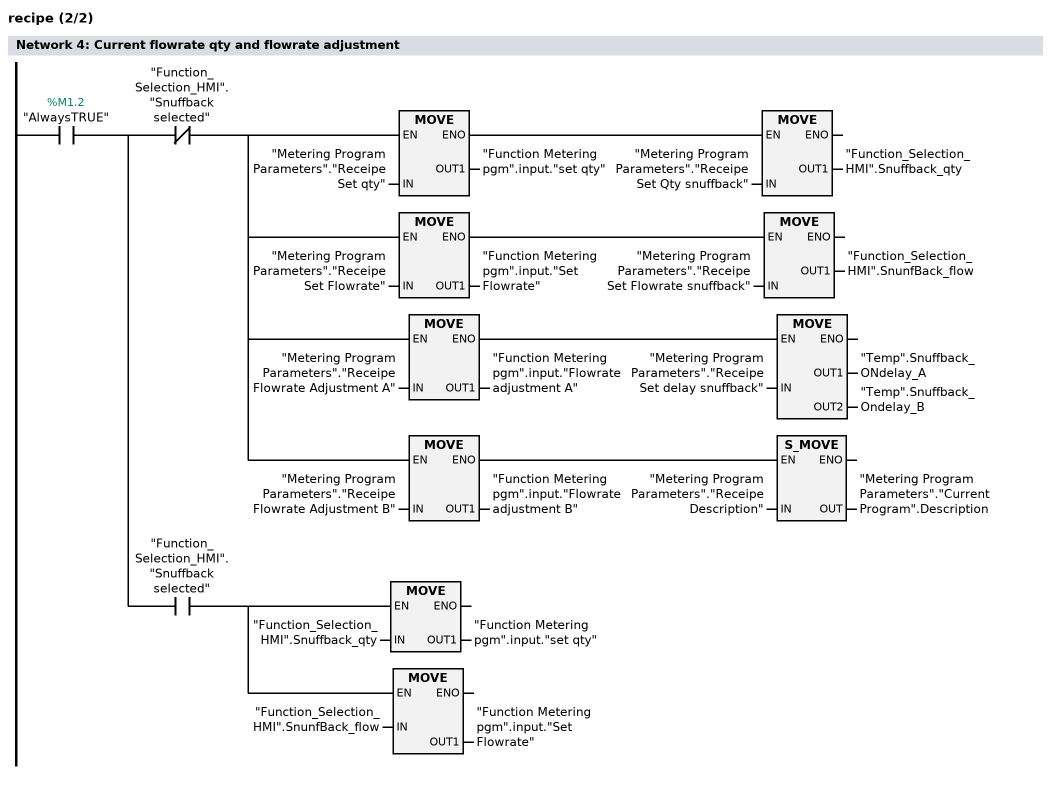
   RUNG wire#powerrail
      Contact( "AlwaysTRUE" )
      wire#w1
      I_Contact( "Function_Selection_HMI"."Snuffback selected" )
      wire#w2
      Move(in := "Metering Program Parameters"."Receipe Set qty", out1 => "Function Metering pgm".input."set qty")
      Move(in := "Metering Program Parameters"."Receipe Set Qty snuffback", out1 => "Function_Selection_HMI".Snuffback_qty)
   END_RUNG
   RUNG wire#w2
      Move(in := "Metering Program Parameters"."Receipe Set Flowrate", out1 => "Function Metering pgm".input."Set Flowrate")
      Move(in := "Metering Program Parameters"."Receipe Set Flowrate snuffback", out1 => "Function_Selection_HMI".SnunfBack_flow)
   END_RUNG
   RUNG wire#w2
      Move(in := "Metering Program Parameters"."Receipe Flowrate Adjustment A", out1 => "Function Metering pgm".input."Flowrate adjustment A")
      Move(in := "Metering Program Parameters"."Receipe Set delay snuffback", out1 => "Temp".Snuffback_ONdelay_A, out2 => "Temp".Snuffback_Ondelay_B)
   END_RUNG
   RUNG wire#w2
      Move(in := "Metering Program Parameters"."Receipe Flowrate Adjustment B", out1 => "Function Metering pgm".input."Flowrate adjustment B")
      S_Move(in := "Metering Program Parameters"."Receipe Description", out => "Metering Program Parameters"."Current Program".Description)
   END_RUNG
   RUNG wire#w1
      Contact( "Function_Selection_HMI"."Snuffback selected" )
      wire#w3
      Move(in := "Function_Selection_HMI".Snuffback_qty, out1 => "Function Metering pgm".input."set qty")
   END_RUNG
   RUNG wire#w3
      Move(in := "Function_Selection_HMI".SnunfBack_flow, out1 => "Function Metering pgm".input."Set Flowrate")
   END_RUNG
   // the same network as SCL:
   IF "AlwaysTRUE" AND NOT "Function_Selection_HMI"."Snuffback selected" THEN
       "Function Metering pgm".input."set qty" := "Metering Program Parameters"."Receipe Set qty";
       "Function_Selection_HMI".Snuffback_qty := "Metering Program Parameters"."Receipe Set Qty snuffback";
       "Function Metering pgm".input."Set Flowrate" := "Metering Program Parameters"."Receipe Set Flowrate";
       "Function_Selection_HMI".SnunfBack_flow := "Metering Program Parameters"."Receipe Set Flowrate snuffback";
       "Function Metering pgm".input."Flowrate adjustment A" := "Metering Program Parameters"."Receipe Flowrate Adjustment A";
       "Temp".Snuffback_ONdelay_A := "Metering Program Parameters"."Receipe Set delay snuffback";
       "Temp".Snuffback_Ondelay_B := "Metering Program Parameters"."Receipe Set delay snuffback";
       "Function Metering pgm".input."Flowrate adjustment B" := "Metering Program Parameters"."Receipe Flowrate Adjustment B";
       "Metering Program Parameters"."Current Program".Description := "Metering Program Parameters"."Receipe Description";
   END_IF;
   IF "AlwaysTRUE" AND "Function_Selection_HMI"."Snuffback selected" THEN
       "Function Metering pgm".input."set qty" := "Function_Selection_HMI".Snuffback_qty;
       "Function Metering pgm".input."Set Flowrate" := "Function_Selection_HMI".SnunfBack_flow;
   END_IF;
END_REGION
END_FUNCTION

FUNCTION "mixing ratio & material Data" : Void   // FC37, LAD
{ S7_Optimized_Access := 'TRUE' }
VERSION : 0.1
// stored: AutoNumber true, IsIECCheckEnabled false, SetENOAutomatically false, UDAEnableTagReadback false
BEGIN

REGION Network 1 (SCL)
   "Material Data current pgm"."name A+B" := CONCAT(IN1 := "Material Data current pgm".Name.A, IN2 :="Material Data current pgm"."+symbol", IN3 := "Material Data current pgm".Name.B);
END_REGION

REGION Network 2: mixing Ratio according to density
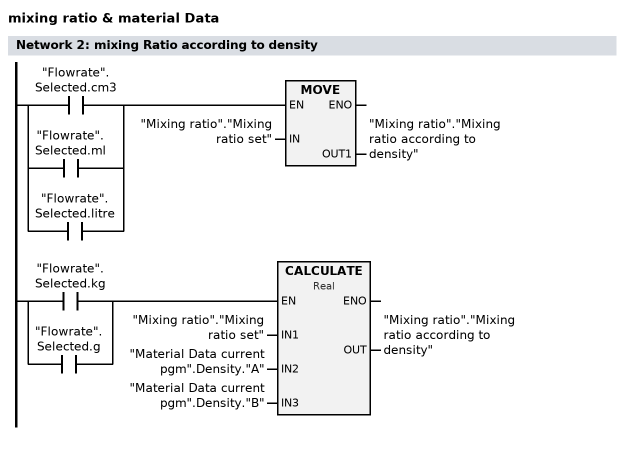
   RUNG wire#powerrail
      Contact( "Flowrate".Selected.cm3 )
      wire#w1
      Move(in := "Mixing ratio"."Mixing ratio set", out1 => "Mixing ratio"."Mixing ratio according to density")
   END_RUNG
   RUNG wire#powerrail
      Contact( "Flowrate".Selected.ml )
   END_RUNG wire#w1
   RUNG wire#powerrail
      Contact( "Flowrate".Selected.litre )
   END_RUNG wire#w1
   RUNG wire#powerrail
      Contact( "Flowrate".Selected.kg )
      wire#w2
      { S7_Templates := "SrcType := Real"; S7_Expression := "(IN1/IN2)*IN3" } Calculate(in1 := "Mixing ratio"."Mixing ratio set", in2 := "Material Data current pgm".Density."A", in3 := "Material Data current pgm".Density."B", out => "Mixing ratio"."Mixing ratio according to density")
   END_RUNG
   RUNG wire#powerrail
      Contact( "Flowrate".Selected.g )
   END_RUNG wire#w2
   // the same network as SCL:
   IF "Flowrate".Selected.cm3 OR "Flowrate".Selected.ml OR "Flowrate".Selected.litre THEN
       "Mixing ratio"."Mixing ratio according to density" := "Mixing ratio"."Mixing ratio set";
   END_IF;
   IF "Flowrate".Selected.kg OR "Flowrate".Selected.g THEN
       "Mixing ratio"."Mixing ratio according to density" := ("Mixing ratio"."Mixing ratio set"/"Material Data current pgm".Density."A")*"Material Data current pgm".Density."B";
   END_IF;
END_REGION
END_FUNCTION

FUNCTION "Operator message1" : Void   // FC29, LAD
{ S7_Optimized_Access := 'TRUE' }
VERSION : 0.1
// stored: AutoNumber true, IsIECCheckEnabled false, SetENOAutomatically false, UDAEnableTagReadback false
BEGIN

REGION Network 1
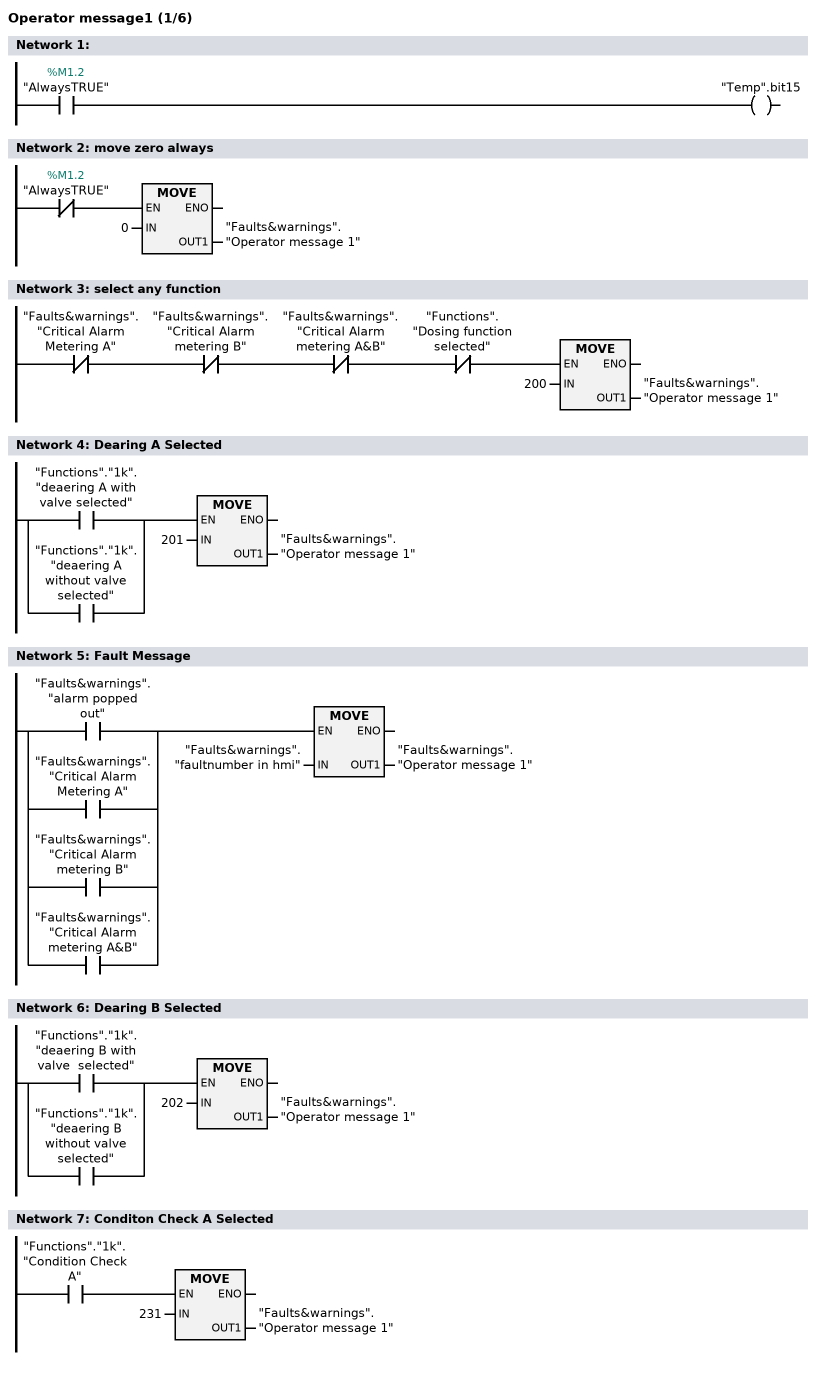
   RUNG wire#powerrail
      Contact( "AlwaysTRUE" )
      Coil( "Temp".bit15 )
   END_RUNG
   // the same network as SCL:
   "Temp".bit15 := "AlwaysTRUE";
END_REGION

REGION Network 2: move zero always
   RUNG wire#powerrail
      I_Contact( "AlwaysTRUE" )
      Move(in := 0, out1 => "Faults&warnings"."Operator message 1")
   END_RUNG
   // the same network as SCL:
   IF NOT "AlwaysTRUE" THEN "Faults&warnings"."Operator message 1" := 0; END_IF;
END_REGION

REGION Network 3: select any function
   RUNG wire#powerrail
      I_Contact( "Faults&warnings"."Critical Alarm Metering A" )
      I_Contact( "Faults&warnings"."Critical Alarm metering B" )
      I_Contact( "Faults&warnings"."Critical Alarm metering A&B" )
      I_Contact( "Functions"."Dosing function selected" )
      Move(in := 200, out1 => "Faults&warnings"."Operator message 1")
   END_RUNG
   // the same network as SCL:
   IF NOT "Faults&warnings"."Critical Alarm Metering A" AND NOT "Faults&warnings"."Critical Alarm metering B" AND NOT "Faults&warnings"."Critical Alarm metering A&B" AND NOT "Functions"."Dosing function selected" THEN
       "Faults&warnings"."Operator message 1" := 200;
   END_IF;
END_REGION

REGION Network 4: Dearing A Selected
   RUNG wire#powerrail
      Contact( "Functions"."1k"."deaering A with valve selected" )
      wire#w1
      Move(in := 201, out1 => "Faults&warnings"."Operator message 1")
   END_RUNG
   RUNG wire#powerrail
      Contact( "Functions"."1k"."deaering A without valve selected" )
   END_RUNG wire#w1
   // the same network as SCL:
   IF "Functions"."1k"."deaering A with valve selected" OR "Functions"."1k"."deaering A without valve selected" THEN
       "Faults&warnings"."Operator message 1" := 201;
   END_IF;
END_REGION

REGION Network 5: Fault Message
   RUNG wire#powerrail
      Contact( "Faults&warnings"."alarm popped out" )
      wire#w1
      Move(in := "Faults&warnings"."faultnumber in hmi", out1 => "Faults&warnings"."Operator message 1")
   END_RUNG
   RUNG wire#powerrail
      Contact( "Faults&warnings"."Critical Alarm Metering A" )
   END_RUNG wire#w1
   RUNG wire#powerrail
      Contact( "Faults&warnings"."Critical Alarm metering B" )
   END_RUNG wire#w1
   RUNG wire#powerrail
      Contact( "Faults&warnings"."Critical Alarm metering A&B" )
   END_RUNG wire#w1
   // the same network as SCL:
   IF "Faults&warnings"."alarm popped out" OR "Faults&warnings"."Critical Alarm Metering A" OR "Faults&warnings"."Critical Alarm metering B" OR "Faults&warnings"."Critical Alarm metering A&B" THEN
       "Faults&warnings"."Operator message 1" := "Faults&warnings"."faultnumber in hmi";
   END_IF;
END_REGION

REGION Network 6: Dearing B Selected
   RUNG wire#powerrail
      Contact( "Functions"."1k"."deaering B with valve  selected" )
      wire#w1
      Move(in := 202, out1 => "Faults&warnings"."Operator message 1")
   END_RUNG
   RUNG wire#powerrail
      Contact( "Functions"."1k"."deaering B without valve  selected" )
   END_RUNG wire#w1
   // the same network as SCL:
   IF "Functions"."1k"."deaering B with valve  selected" OR "Functions"."1k"."deaering B without valve  selected" THEN
       "Faults&warnings"."Operator message 1" := 202;
   END_IF;
END_REGION

REGION Network 7: Conditon Check A Selected
   RUNG wire#powerrail
      Contact( "Functions"."1k"."Condition Check A" )
      Move(in := 231, out1 => "Faults&warnings"."Operator message 1")
   END_RUNG
   // the same network as SCL:
   IF "Functions"."1k"."Condition Check A" THEN "Faults&warnings"."Operator message 1" := 231; END_IF;
END_REGION

REGION Network 8: Conditon Check B Selected
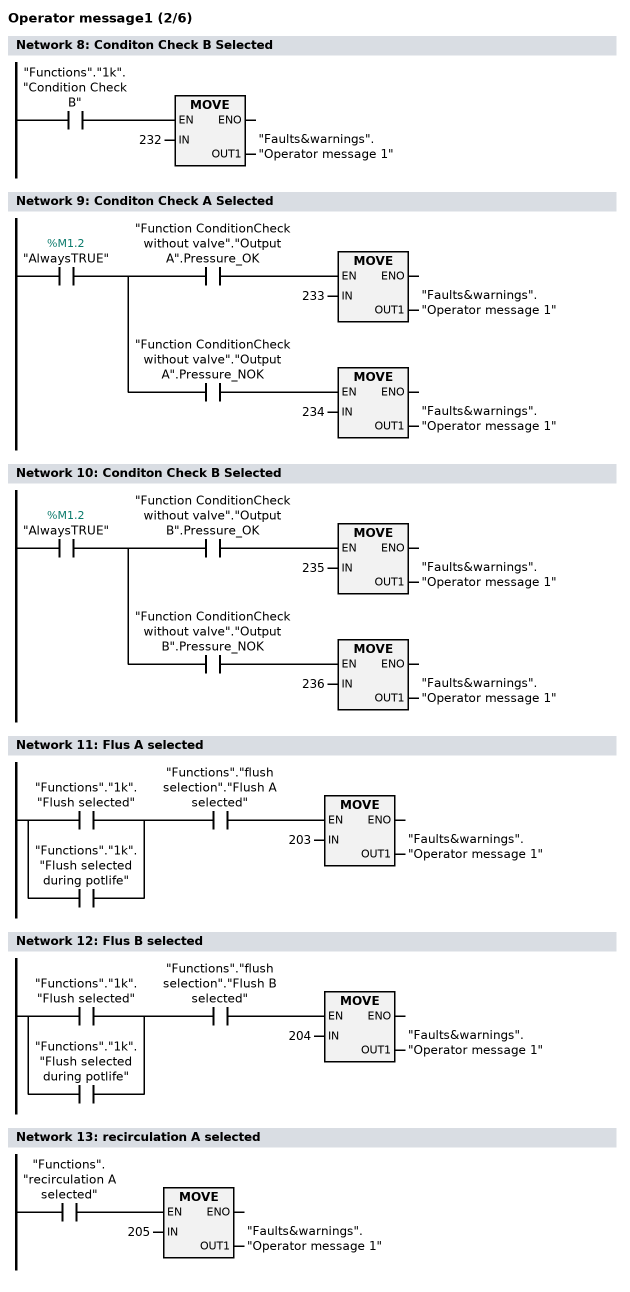
   RUNG wire#powerrail
      Contact( "Functions"."1k"."Condition Check B" )
      Move(in := 232, out1 => "Faults&warnings"."Operator message 1")
   END_RUNG
   // the same network as SCL:
   IF "Functions"."1k"."Condition Check B" THEN "Faults&warnings"."Operator message 1" := 232; END_IF;
END_REGION

REGION Network 9: Conditon Check A Selected
   RUNG wire#powerrail
      Contact( "AlwaysTRUE" )
      wire#w1
      Contact( "Function ConditionCheck without valve"."Output A".Pressure_OK )
      Move(in := 233, out1 => "Faults&warnings"."Operator message 1")
   END_RUNG
   RUNG wire#w1
      Contact( "Function ConditionCheck without valve"."Output A".Pressure_NOK )
      Move(in := 234, out1 => "Faults&warnings"."Operator message 1")
   END_RUNG
   // the same network as SCL:
   IF "AlwaysTRUE" AND "Function ConditionCheck without valve"."Output A".Pressure_OK THEN
       "Faults&warnings"."Operator message 1" := 233;
   END_IF;
   IF "AlwaysTRUE" AND "Function ConditionCheck without valve"."Output A".Pressure_NOK THEN
       "Faults&warnings"."Operator message 1" := 234;
   END_IF;
END_REGION

REGION Network 10: Conditon Check B Selected
   RUNG wire#powerrail
      Contact( "AlwaysTRUE" )
      wire#w1
      Contact( "Function ConditionCheck without valve"."Output B".Pressure_OK )
      Move(in := 235, out1 => "Faults&warnings"."Operator message 1")
   END_RUNG
   RUNG wire#w1
      Contact( "Function ConditionCheck without valve"."Output B".Pressure_NOK )
      Move(in := 236, out1 => "Faults&warnings"."Operator message 1")
   END_RUNG
   // the same network as SCL:
   IF "AlwaysTRUE" AND "Function ConditionCheck without valve"."Output B".Pressure_OK THEN
       "Faults&warnings"."Operator message 1" := 235;
   END_IF;
   IF "AlwaysTRUE" AND "Function ConditionCheck without valve"."Output B".Pressure_NOK THEN
       "Faults&warnings"."Operator message 1" := 236;
   END_IF;
END_REGION

REGION Network 11: Flus A selected
   RUNG wire#powerrail
      Contact( "Functions"."1k"."Flush selected" )
      wire#w1
      Contact( "Functions"."flush selection"."Flush A selected" )
      Move(in := 203, out1 => "Faults&warnings"."Operator message 1")
   END_RUNG
   RUNG wire#powerrail
      Contact( "Functions"."1k"."Flush selected during potlife" )
   END_RUNG wire#w1
   // the same network as SCL:
   IF ("Functions"."1k"."Flush selected" OR "Functions"."1k"."Flush selected during potlife") AND "Functions"."flush selection"."Flush A selected" THEN
       "Faults&warnings"."Operator message 1" := 203;
   END_IF;
END_REGION

REGION Network 12: Flus B selected
   RUNG wire#powerrail
      Contact( "Functions"."1k"."Flush selected" )
      wire#w1
      Contact( "Functions"."flush selection"."Flush B selected" )
      Move(in := 204, out1 => "Faults&warnings"."Operator message 1")
   END_RUNG
   RUNG wire#powerrail
      Contact( "Functions"."1k"."Flush selected during potlife" )
   END_RUNG wire#w1
   // the same network as SCL:
   IF ("Functions"."1k"."Flush selected" OR "Functions"."1k"."Flush selected during potlife") AND "Functions"."flush selection"."Flush B selected" THEN
       "Faults&warnings"."Operator message 1" := 204;
   END_IF;
END_REGION

REGION Network 13: recirculation A selected
   RUNG wire#powerrail
      Contact( "Functions"."recirculation A selected" )
      Move(in := 205, out1 => "Faults&warnings"."Operator message 1")
   END_RUNG
   // the same network as SCL:
   IF "Functions"."recirculation A selected" THEN "Faults&warnings"."Operator message 1" := 205; END_IF;
END_REGION

REGION Network 14: recirculation B selected
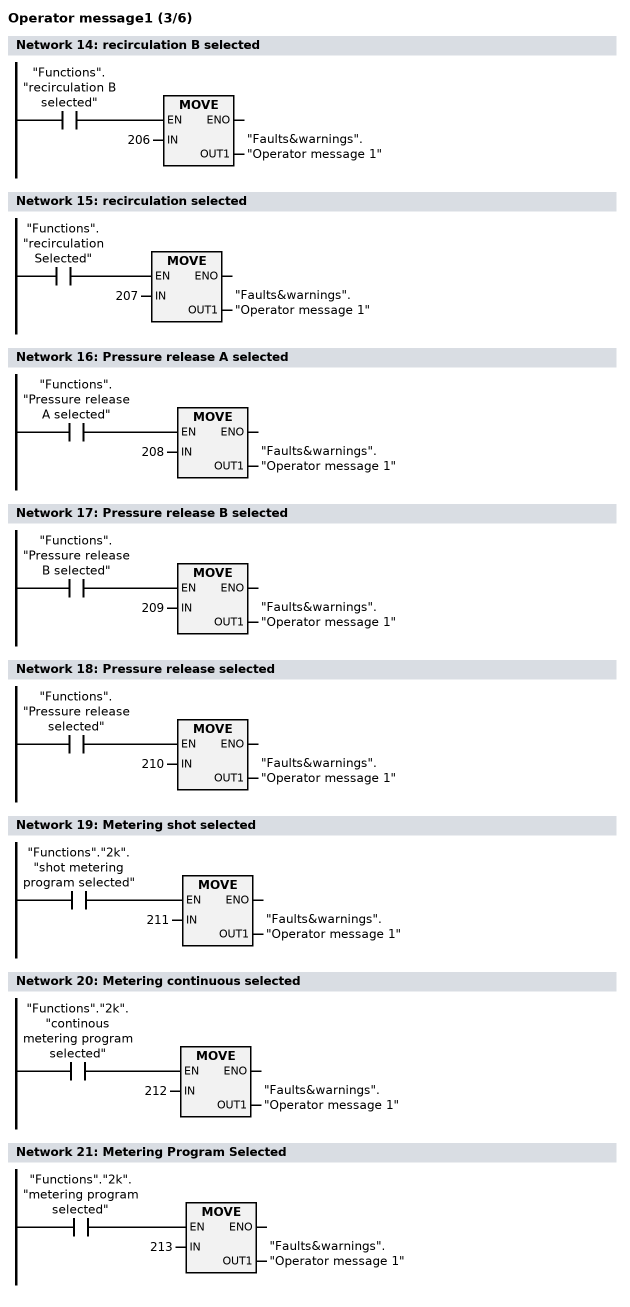
   RUNG wire#powerrail
      Contact( "Functions"."recirculation B selected" )
      Move(in := 206, out1 => "Faults&warnings"."Operator message 1")
   END_RUNG
   // the same network as SCL:
   IF "Functions"."recirculation B selected" THEN "Faults&warnings"."Operator message 1" := 206; END_IF;
END_REGION

REGION Network 15: recirculation selected
   RUNG wire#powerrail
      Contact( "Functions"."recirculation Selected" )
      Move(in := 207, out1 => "Faults&warnings"."Operator message 1")
   END_RUNG
   // the same network as SCL:
   IF "Functions"."recirculation Selected" THEN "Faults&warnings"."Operator message 1" := 207; END_IF;
END_REGION

REGION Network 16: Pressure release A selected
   RUNG wire#powerrail
      Contact( "Functions"."Pressure release A selected" )
      Move(in := 208, out1 => "Faults&warnings"."Operator message 1")
   END_RUNG
   // the same network as SCL:
   IF "Functions"."Pressure release A selected" THEN "Faults&warnings"."Operator message 1" := 208; END_IF;
END_REGION

REGION Network 17: Pressure release B selected
   RUNG wire#powerrail
      Contact( "Functions"."Pressure release B selected" )
      Move(in := 209, out1 => "Faults&warnings"."Operator message 1")
   END_RUNG
   // the same network as SCL:
   IF "Functions"."Pressure release B selected" THEN "Faults&warnings"."Operator message 1" := 209; END_IF;
END_REGION

REGION Network 18: Pressure release selected
   RUNG wire#powerrail
      Contact( "Functions"."Pressure release selected" )
      Move(in := 210, out1 => "Faults&warnings"."Operator message 1")
   END_RUNG
   // the same network as SCL:
   IF "Functions"."Pressure release selected" THEN "Faults&warnings"."Operator message 1" := 210; END_IF;
END_REGION

REGION Network 19: Metering shot selected
   RUNG wire#powerrail
      Contact( "Functions"."2k"."shot metering program selected" )
      Move(in := 211, out1 => "Faults&warnings"."Operator message 1")
   END_RUNG
   // the same network as SCL:
   IF "Functions"."2k"."shot metering program selected" THEN
       "Faults&warnings"."Operator message 1" := 211;
   END_IF;
END_REGION

REGION Network 20: Metering continuous selected
   RUNG wire#powerrail
      Contact( "Functions"."2k"."continous metering program selected" )
      Move(in := 212, out1 => "Faults&warnings"."Operator message 1")
   END_RUNG
   // the same network as SCL:
   IF "Functions"."2k"."continous metering program selected" THEN
       "Faults&warnings"."Operator message 1" := 212;
   END_IF;
END_REGION

REGION Network 21: Metering Program Selected
   RUNG wire#powerrail
      Contact( "Functions"."2k"."metering program selected" )
      Move(in := 213, out1 => "Faults&warnings"."Operator message 1")
   END_RUNG
   // the same network as SCL:
   IF "Functions"."2k"."metering program selected" THEN
       "Faults&warnings"."Operator message 1" := 213;
   END_IF;
END_REGION

REGION Network 22: Pre run Program Selected
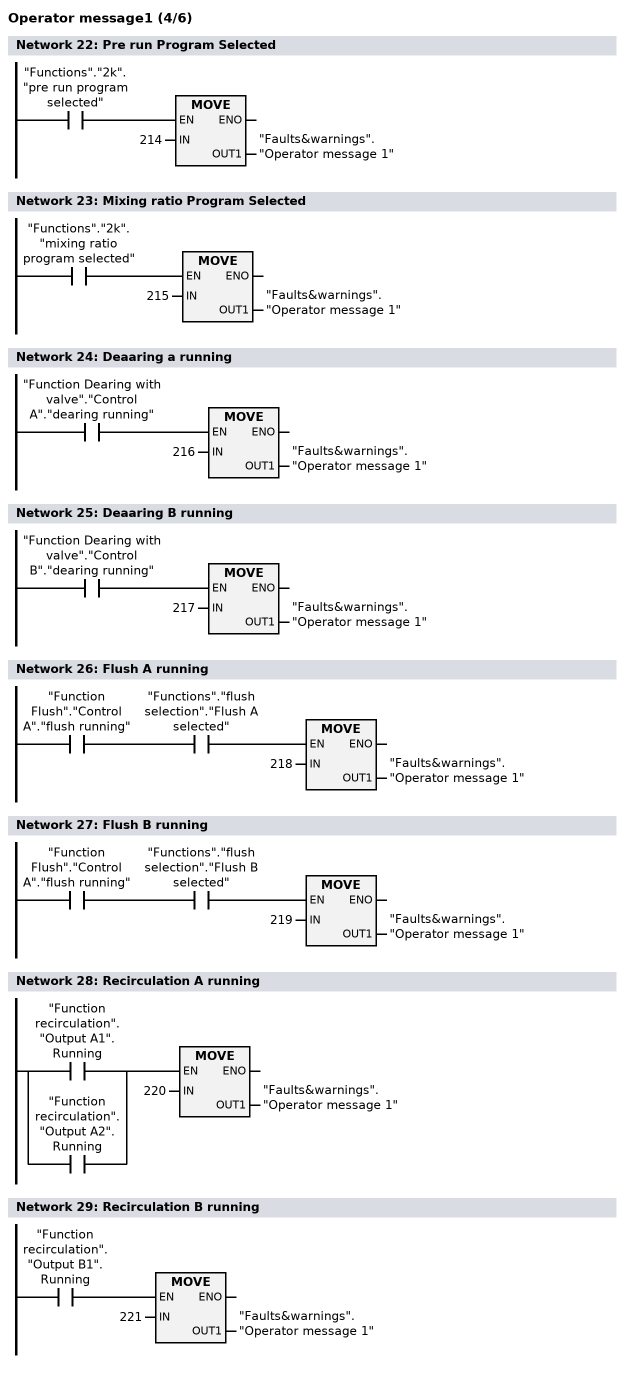
   RUNG wire#powerrail
      Contact( "Functions"."2k"."pre run program selected" )
      Move(in := 214, out1 => "Faults&warnings"."Operator message 1")
   END_RUNG
   // the same network as SCL:
   IF "Functions"."2k"."pre run program selected" THEN "Faults&warnings"."Operator message 1" := 214; END_IF;
END_REGION

REGION Network 23: Mixing ratio Program Selected
   RUNG wire#powerrail
      Contact( "Functions"."2k"."mixing ratio program selected" )
      Move(in := 215, out1 => "Faults&warnings"."Operator message 1")
   END_RUNG
   // the same network as SCL:
   IF "Functions"."2k"."mixing ratio program selected" THEN
       "Faults&warnings"."Operator message 1" := 215;
   END_IF;
END_REGION

REGION Network 24: Deaaring a running
   RUNG wire#powerrail
      Contact( "Function Dearing with valve"."Control A"."dearing running" )
      Move(in := 216, out1 => "Faults&warnings"."Operator message 1")
   END_RUNG
   // the same network as SCL:
   IF "Function Dearing with valve"."Control A"."dearing running" THEN
       "Faults&warnings"."Operator message 1" := 216;
   END_IF;
END_REGION

REGION Network 25: Deaaring B running
   RUNG wire#powerrail
      Contact( "Function Dearing with valve"."Control B"."dearing running" )
      Move(in := 217, out1 => "Faults&warnings"."Operator message 1")
   END_RUNG
   // the same network as SCL:
   IF "Function Dearing with valve"."Control B"."dearing running" THEN
       "Faults&warnings"."Operator message 1" := 217;
   END_IF;
END_REGION

REGION Network 26: Flush A running
   RUNG wire#powerrail
      Contact( "Function Flush"."Control A"."flush running" )
      Contact( "Functions"."flush selection"."Flush A selected" )
      Move(in := 218, out1 => "Faults&warnings"."Operator message 1")
   END_RUNG
   // the same network as SCL:
   IF "Function Flush"."Control A"."flush running" AND "Functions"."flush selection"."Flush A selected" THEN
       "Faults&warnings"."Operator message 1" := 218;
   END_IF;
END_REGION

REGION Network 27: Flush B running
   RUNG wire#powerrail
      Contact( "Function Flush"."Control A"."flush running" )
      Contact( "Functions"."flush selection"."Flush B selected" )
      Move(in := 219, out1 => "Faults&warnings"."Operator message 1")
   END_RUNG
   // the same network as SCL:
   IF "Function Flush"."Control A"."flush running" AND "Functions"."flush selection"."Flush B selected" THEN
       "Faults&warnings"."Operator message 1" := 219;
   END_IF;
END_REGION

REGION Network 28: Recirculation A running
   RUNG wire#powerrail
      Contact( "Function recirculation"."Output A1".Running )
      wire#w1
      Move(in := 220, out1 => "Faults&warnings"."Operator message 1")
   END_RUNG
   RUNG wire#powerrail
      Contact( "Function recirculation"."Output A2".Running )
   END_RUNG wire#w1
   // the same network as SCL:
   IF "Function recirculation"."Output A1".Running OR "Function recirculation"."Output A2".Running THEN
       "Faults&warnings"."Operator message 1" := 220;
   END_IF;
END_REGION

REGION Network 29: Recirculation B running
   RUNG wire#powerrail
      Contact( "Function recirculation"."Output B1".Running )
      Move(in := 221, out1 => "Faults&warnings"."Operator message 1")
   END_RUNG
   // the same network as SCL:
   IF "Function recirculation"."Output B1".Running THEN
       "Faults&warnings"."Operator message 1" := 221;
   END_IF;
END_REGION

REGION Network 30: Recirculation running
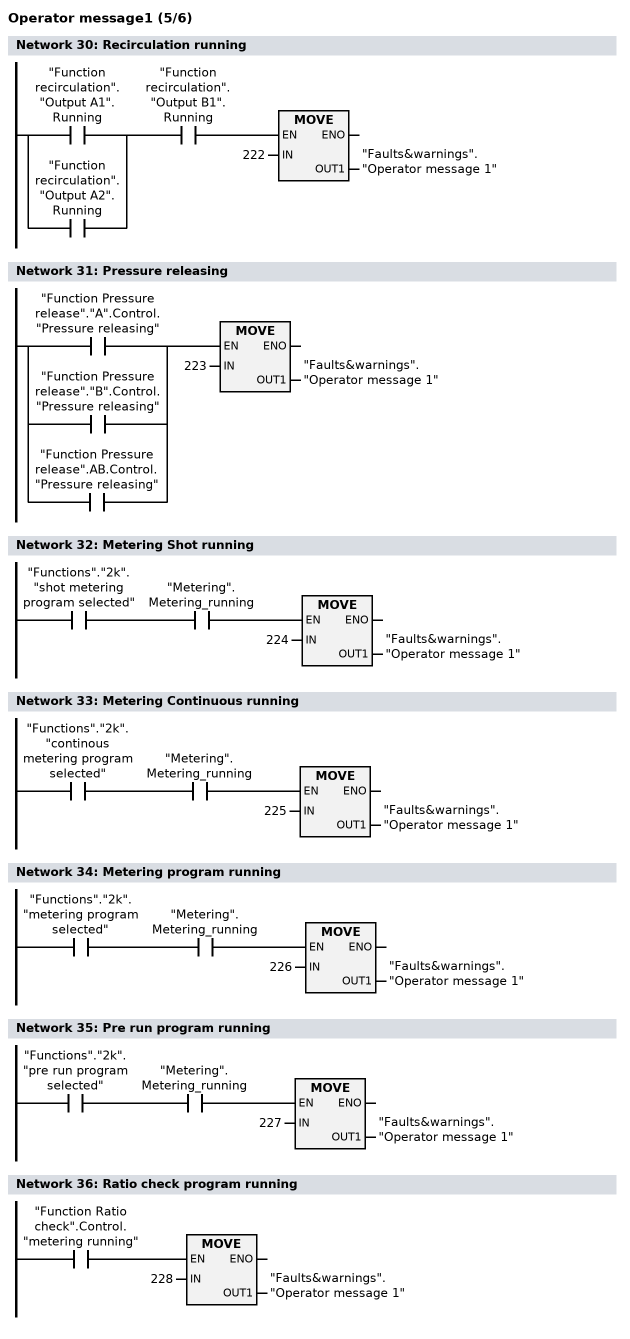
   RUNG wire#powerrail
      Contact( "Function recirculation"."Output A1".Running )
      wire#w1
      Contact( "Function recirculation"."Output B1".Running )
      Move(in := 222, out1 => "Faults&warnings"."Operator message 1")
   END_RUNG
   RUNG wire#powerrail
      Contact( "Function recirculation"."Output A2".Running )
   END_RUNG wire#w1
   // the same network as SCL:
   IF ("Function recirculation"."Output A1".Running OR "Function recirculation"."Output A2".Running) AND "Function recirculation"."Output B1".Running THEN
       "Faults&warnings"."Operator message 1" := 222;
   END_IF;
END_REGION

REGION Network 31: Pressure releasing
   RUNG wire#powerrail
      Contact( "Function Pressure release"."A".Control."Pressure releasing" )
      wire#w1
      Move(in := 223, out1 => "Faults&warnings"."Operator message 1")
   END_RUNG
   RUNG wire#powerrail
      Contact( "Function Pressure release"."B".Control."Pressure releasing" )
   END_RUNG wire#w1
   RUNG wire#powerrail
      Contact( "Function Pressure release".AB.Control."Pressure releasing" )
   END_RUNG wire#w1
   // the same network as SCL:
   IF "Function Pressure release"."A".Control."Pressure releasing" OR "Function Pressure release"."B".Control."Pressure releasing" OR "Function Pressure release".AB.Control."Pressure releasing" THEN
       "Faults&warnings"."Operator message 1" := 223;
   END_IF;
END_REGION

REGION Network 32: Metering Shot running
   RUNG wire#powerrail
      Contact( "Functions"."2k"."shot metering program selected" )
      Contact( "Metering".Metering_running )
      Move(in := 224, out1 => "Faults&warnings"."Operator message 1")
   END_RUNG
   // the same network as SCL:
   IF "Functions"."2k"."shot metering program selected" AND "Metering".Metering_running THEN
       "Faults&warnings"."Operator message 1" := 224;
   END_IF;
END_REGION

REGION Network 33: Metering Continuous running
   RUNG wire#powerrail
      Contact( "Functions"."2k"."continous metering program selected" )
      Contact( "Metering".Metering_running )
      Move(in := 225, out1 => "Faults&warnings"."Operator message 1")
   END_RUNG
   // the same network as SCL:
   IF "Functions"."2k"."continous metering program selected" AND "Metering".Metering_running THEN
       "Faults&warnings"."Operator message 1" := 225;
   END_IF;
END_REGION

REGION Network 34: Metering program running
   RUNG wire#powerrail
      Contact( "Functions"."2k"."metering program selected" )
      Contact( "Metering".Metering_running )
      Move(in := 226, out1 => "Faults&warnings"."Operator message 1")
   END_RUNG
   // the same network as SCL:
   IF "Functions"."2k"."metering program selected" AND "Metering".Metering_running THEN
       "Faults&warnings"."Operator message 1" := 226;
   END_IF;
END_REGION

REGION Network 35: Pre run program running
   RUNG wire#powerrail
      Contact( "Functions"."2k"."pre run program selected" )
      Contact( "Metering".Metering_running )
      Move(in := 227, out1 => "Faults&warnings"."Operator message 1")
   END_RUNG
   // the same network as SCL:
   IF "Functions"."2k"."pre run program selected" AND "Metering".Metering_running THEN
       "Faults&warnings"."Operator message 1" := 227;
   END_IF;
END_REGION

REGION Network 36: Ratio check program running
   RUNG wire#powerrail
      Contact( "Function Ratio check".Control."metering running" )
      Move(in := 228, out1 => "Faults&warnings"."Operator message 1")
   END_RUNG
   // the same network as SCL:
   IF "Function Ratio check".Control."metering running" THEN
       "Faults&warnings"."Operator message 1" := 228;
   END_IF;
END_REGION

REGION Network 37: Reneration program Selected
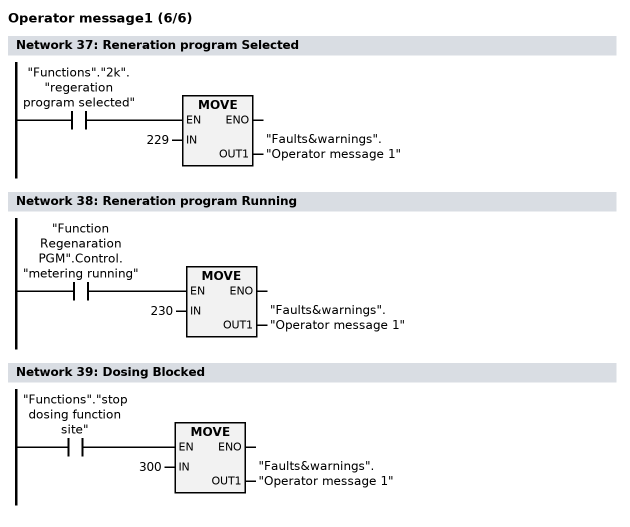
   RUNG wire#powerrail
      Contact( "Functions"."2k"."regeration program selected" )
      Move(in := 229, out1 => "Faults&warnings"."Operator message 1")
   END_RUNG
   // the same network as SCL:
   IF "Functions"."2k"."regeration program selected" THEN
       "Faults&warnings"."Operator message 1" := 229;
   END_IF;
END_REGION

REGION Network 38: Reneration program Running
   RUNG wire#powerrail
      Contact( "Function Regenaration PGM".Control."metering running" )
      Move(in := 230, out1 => "Faults&warnings"."Operator message 1")
   END_RUNG
   // the same network as SCL:
   IF "Function Regenaration PGM".Control."metering running" THEN
       "Faults&warnings"."Operator message 1" := 230;
   END_IF;
END_REGION

REGION Network 39: Dosing Blocked
   RUNG wire#powerrail
      Contact( "Functions"."stop dosing function site" )
      Move(in := 300, out1 => "Faults&warnings"."Operator message 1")
   END_RUNG
   // the same network as SCL:
   IF "Functions"."stop dosing function site" THEN "Faults&warnings"."Operator message 1" := 300; END_IF;
END_REGION

REGION Network 40 (SCL)
   // IF "Faults&warnings"."Status Nok"."Low level A1"  THEN
   //   "Faults&warnings"."Operator message 1" := 74;
   // END_IF;
   // IF "Faults&warnings"."Status Nok"."Low level B1" THEN
   //   "Faults&warnings"."Operator message 1" := 75;
   // END_IF;
   // IF "Alarm_DB".input.alarm[21] THEN
   //   "Faults&warnings"."Operator message 1" := 76;
   // END_IF;
   // IF "Alarm_DB".input.alarm[20] THEN
   //     "Faults&warnings"."Operator message 1" := 77;
   // END_IF;

   // IF "Faults&warnings"."Status Nok"."Level Low Drum A1" THEN
   //   "Faults&warnings"."Operator message 1" := 82;
   // END_IF;
   // IF "Faults&warnings"."Status Nok"."Level Low Drum B1" THEN
   //   "Faults&warnings"."Operator message 1" := 83;
   // END_IF;
   // IF "Faults&warnings"."Status Nok"."Level Low Drum A2" THEN
   //   "Faults&warnings"."Operator message 1" := 84;
   // END_IF;
   // IF "Faults&warnings"."Status Nok"."Level Low Drum B2" THEN
   //   "Faults&warnings"."Operator message 1" := 85;
   // END_IF;
   // IF "Faults&warnings"."Status Nok"."Level Empty Drum A1" THEN
   //   "Faults&warnings"."Operator message 1" := 86;
   // END_IF;
   // IF "Faults&warnings"."Status Nok"."Level Empty Drum B1" THEN
   //   "Faults&warnings"."Operator message 1" := 87;
   // END_IF;
   // IF "Faults&warnings"."Status Nok"."Level Empty Drum A2" THEN
   //   "Faults&warnings"."Operator message 1" := 88;
   // END_IF;
   // IF "Faults&warnings"."Status Nok"."Level Empty Drum B2" THEN
   //   "Faults&warnings"."Operator message 1" := 89;
   // END_IF;
END_REGION
END_FUNCTION

FUNCTION "Operator message 2" : Void   // FC33, LAD
{ S7_Optimized_Access := 'TRUE' }
VERSION : 0.1
// stored: AutoNumber true, IsIECCheckEnabled false, SetENOAutomatically false, UDAEnableTagReadback false
BEGIN

REGION Network 1 (SCL)
   IF "Faults&warnings"."Critical Alarm Metering A" OR "Faults&warnings"."Critical Alarm metering B" OR "Faults&warnings"."Critical Alarm metering A&B" THEN
       "Faults&warnings"."Operator message 2" := 8; // Machine error
   ELSIF "Functions"."stop dosing function site" THEN
       "Faults&warnings"."Operator message 2" := 7; // Metering blocked
   ELSIF "Functions"."Dosing function selected" AND
       ("Faults&warnings"."Critical Alarm Metering A" OR "Faults&warnings"."Critical Alarm metering B" OR "Faults&warnings"."Critical Alarm metering A&B") THEN
       "Faults&warnings"."Operator message 2" := 6; // Metering blocked
   ELSIF "Functions"."Dosing function selected" AND "Functions"."Dosing Running" AND "Function_Selection_HMI"."Snuffback selected" AND
       ("Function_Selection_HMI".Function_Snuffback_volume_dispensed < "Function_Selection_HMI".Snuffback_qty) THEN
       "Faults&warnings"."Operator message 2" := 9;
   ELSIF "Functions"."Dosing function selected" AND "Functions"."Dosing Running" AND NOT ("Function_Selection_HMI"."Snuffback selected") THEN
       "Faults&warnings"."Operator message 2" := 5; //function running
   ELSIF "Control"."waiting For pre run" AND NOT ("Functions"."Dosing function selected") THEN
       "Faults&warnings"."Operator message 2" := 4; // waiting for prerun   
   ELSIF "Functions"."Dosing function selected" AND NOT ("Pump & Flowrate".startSnuff_Back_PumpA) AND NOT ("Pump & Flowrate".startSnuff_Back_PumpB) THEN
       "Faults&warnings"."Operator message 2" := 3; // waiting for start\
   ELSIF "Control"."waiting For pre run" = false THEN
       "Faults&warnings"."Operator message 2" := 2; // ready for operation
   ELSIF     "Faults&warnings"."Fault present" = false THEN
       "Faults&warnings"."Operator message 2" := 1; // machnie ready

   END_IF;
END_REGION
END_FUNCTION

FUNCTION "Output" : Void   // FC32, LAD
{ S7_Optimized_Access := 'TRUE' }
VERSION : 0.1
// stored: AutoNumber true, IsIECCheckEnabled false, SetENOAutomatically false, UDAEnableTagReadback false
BEGIN

REGION Network 1: tower lamp amber
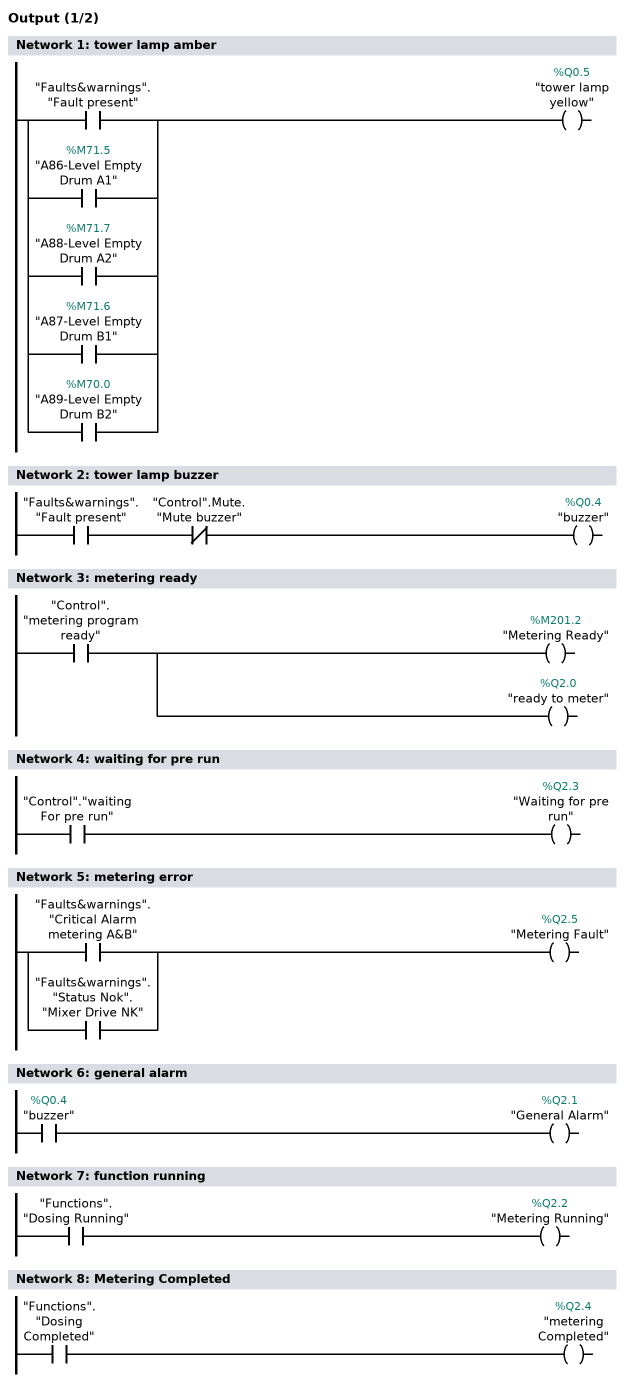
   RUNG wire#powerrail
      Contact( "Faults&warnings"."Fault present" )
      wire#w1
      Coil( "tower lamp yellow" )
   END_RUNG
   RUNG wire#powerrail
      Contact( "A86-Level Empty Drum A1" )
   END_RUNG wire#w1
   RUNG wire#powerrail
      Contact( "A88-Level Empty Drum A2" )
   END_RUNG wire#w1
   RUNG wire#powerrail
      Contact( "A87-Level Empty Drum B1" )
   END_RUNG wire#w1
   RUNG wire#powerrail
      Contact( "A89-Level Empty Drum B2" )
   END_RUNG wire#w1
   // the same network as SCL:
   "tower lamp yellow" := "Faults&warnings"."Fault present" OR "A86-Level Empty Drum A1" OR "A88-Level Empty Drum A2" OR "A87-Level Empty Drum B1" OR "A89-Level Empty Drum B2";
END_REGION

REGION Network 2: tower lamp buzzer
   RUNG wire#powerrail
      Contact( "Faults&warnings"."Fault present" )
      I_Contact( "Control".Mute."Mute buzzer" )
      Coil( "buzzer" )
   END_RUNG
   // the same network as SCL:
   "buzzer" := "Faults&warnings"."Fault present" AND NOT "Control".Mute."Mute buzzer";
END_REGION

REGION Network 3: metering ready
   RUNG wire#powerrail
      Contact( "Control"."metering program ready" )
      wire#w1
      Coil( "Metering Ready" )
   END_RUNG
   RUNG wire#w1
      Coil( "ready to meter" )
   END_RUNG
   // the same network as SCL:
   "Metering Ready" := "Control"."metering program ready";
   "ready to meter" := "Control"."metering program ready";
END_REGION

REGION Network 4: waiting for pre run
   RUNG wire#powerrail
      Contact( "Control"."waiting For pre run" )
      Coil( "Waiting for pre run" )
   END_RUNG
   // the same network as SCL:
   "Waiting for pre run" := "Control"."waiting For pre run";
END_REGION

REGION Network 5: metering error
   RUNG wire#powerrail
      Contact( "Faults&warnings"."Critical Alarm metering A&B" )
      wire#w1
      Coil( "Metering Fault" )
   END_RUNG
   RUNG wire#powerrail
      Contact( "Faults&warnings"."Status Nok"."Mixer Drive NK" )
   END_RUNG wire#w1
   // the same network as SCL:
   "Metering Fault" := "Faults&warnings"."Critical Alarm metering A&B" OR "Faults&warnings"."Status Nok"."Mixer Drive NK";
END_REGION

REGION Network 6: general alarm
   RUNG wire#powerrail
      Contact( "buzzer" )
      Coil( "General Alarm" )
   END_RUNG
   // the same network as SCL:
   "General Alarm" := "buzzer";
END_REGION

REGION Network 7: function running
   RUNG wire#powerrail
      Contact( "Functions"."Dosing Running" )
      Coil( "Metering Running" )
   END_RUNG
   // the same network as SCL:
   "Metering Running" := "Functions"."Dosing Running";
END_REGION

REGION Network 8: Metering Completed
   RUNG wire#powerrail
      Contact( "Functions"."Dosing Completed" )
      Coil( "metering Completed" )
   END_RUNG
   // the same network as SCL:
   "metering Completed" := "Functions"."Dosing Completed";
END_REGION

REGION Network 9: Control On Lamp
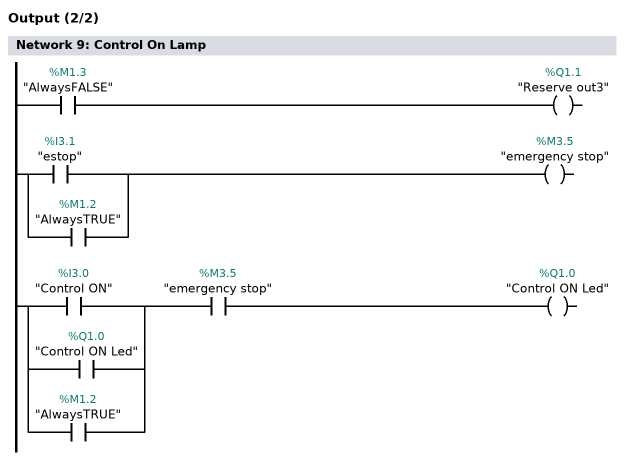
   RUNG wire#powerrail
      Contact( "AlwaysFALSE" )
      Coil( "Reserve out3" )
   END_RUNG
   RUNG wire#powerrail
      Contact( "estop" )
      wire#w1
      Coil( "emergency stop" )
   END_RUNG
   RUNG wire#powerrail
      Contact( "AlwaysTRUE" )
   END_RUNG wire#w1
   RUNG wire#powerrail
      Contact( "Control ON" )
      wire#w2
      Contact( "emergency stop" )
      Coil( "Control ON Led" )
   END_RUNG
   RUNG wire#powerrail
      Contact( "Control ON Led" )
   END_RUNG wire#w2
   RUNG wire#powerrail
      Contact( "AlwaysTRUE" )
   END_RUNG wire#w2
   // the same network as SCL:
   "Reserve out3" := "AlwaysFALSE";
   "emergency stop" := "estop" OR "AlwaysTRUE";
   "Control ON Led" := ("Control ON" OR "Control ON Led" OR "AlwaysTRUE") AND "emergency stop";
END_REGION
END_FUNCTION

FUNCTION "Datalog" : Void   // FC13, LAD
{ S7_Optimized_Access := 'TRUE' }
VERSION : 0.1
// stored: AutoNumber true, IsIECCheckEnabled false, SetENOAutomatically false, UDAEnableTagReadback false
   VAR_TEMP
      "return" : Int;
   END_VAR
   VAR_TEMP   // added for the SCL form of the ladder/FBD networks
      _w1 : Bool;
      _w2 : Bool;
      _w3 : Bool;
      _w4 : Bool;
      _w5 : Bool;
      _w6 : Bool;
      _w7 : Bool;
      _w8 : Bool;
   END_VAR
BEGIN

REGION Network 1
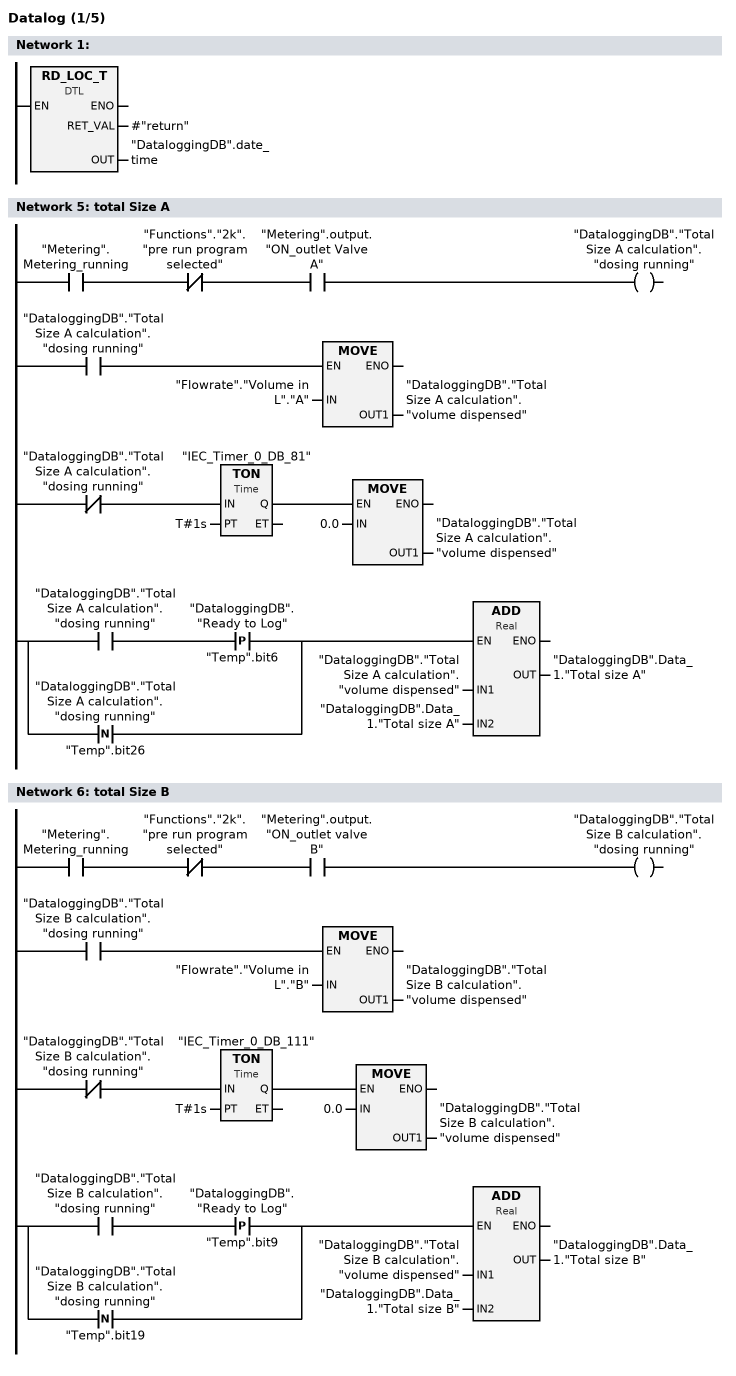
   RUNG wire#powerrail
      { S7_Templates := "date_type := DTL" } RD_LOC_T(RET_VAL => #"return", OUT => "DataloggingDB".date_time)
   END_RUNG
   // the same network as SCL:
   #"return" := RD_LOC_T(OUT => "DataloggingDB".date_time);
END_REGION

REGION Network 2 (SCL)
   IF "DataloggingDB".date_time.DAY <> "DataloggingDB".previous_day THEN
       //"DataloggingDB".day_changed := true;
       "DataloggingDB".totalsizepreviousday:="DataloggingDB".Data_1."Total Size";
       "DataloggingDB".previous_day := "DataloggingDB".date_time.DAY ;
   ELSE
       "DataloggingDB".day_changed := false;
   END_IF;
   IF "DataloggingDB".current_week <> "DataloggingDB".previous_week THEN
       //"DataloggingDB".day_changed := true;
       "DataloggingDB".totalsizepreviousweek := "DataloggingDB".Data_1."Total Size";
       "DataloggingDB".previous_week := "DataloggingDB".current_week;
   ELSE
       "DataloggingDB".day_changed := false;
   END_IF;

   IF "DataloggingDB".date_time.MONTH <> "DataloggingDB".previous_month THEN
       //"DataloggingDB".month_changed := true;
       "DataloggingDB".totalsizepreviousmonth := "DataloggingDB".Data_1."Total Size";
       "DataloggingDB".previous_month := "DataloggingDB".date_time.MONTH;
   ELSE
       "DataloggingDB".month_changed := false;
   END_IF;

   "DataloggingDB".totalsizeday := "DataloggingDB".Data_1."Total Size" - "DataloggingDB".totalsizepreviousday ;
   "DataloggingDB".totalsizeweek := "DataloggingDB".Data_1."Total Size" - "DataloggingDB".totalsizepreviousweek;
   "DataloggingDB".totalsizemonth := "DataloggingDB".Data_1."Total Size" - "DataloggingDB".totalsizepreviousmonth;
END_REGION

REGION Network 3 (SCL): Total Flush A
   IF (("Function Flush"."Control A"."flush running" AND "Functions"."flush selection"."Flush A selected") OR
       "Function Regenaration PGM".Control."metering running" OR
       "Function Ratio check".Control."metering running" OR
       ("Functions"."2k"."pre run program selected" AND "Metering".Metering_running) OR
       "Function Dearing with valve"."Control A"."dearing running") THEN
       "DataloggingDB"."Copy Flush A qty" := true;
   END_IF;

   "R_TRIG_DB_1"(CLK:="DataloggingDB"."Copy Flush A qty" AND NOT ("Function Dearing with valve"."Control A"."dearing running") AND
                 NOT ("Function Regenaration PGM".Control."metering running") AND NOT ("Function Ratio check".Control."metering running") AND
                 NOT ("Functions"."2k"."pre run program selected") AND NOT ("Function Flush"."Control A"."flush running"),
                 Q=>"Temp".bit1);

   IF "R_TRIG_DB_1".Q THEN
       "DataloggingDB".Data_1."Total A flush" := "Flowrate"."Volume in L".mixed +"DataloggingDB".Data_1."Total A flush";
       "DataloggingDB"."Copy Flush A qty" := false;
   END_IF;
END_REGION

REGION Network 4 (SCL)
   IF (("Function Flush"."Control B"."flush running" AND "Functions"."flush selection"."Flush B selected") OR
       "Function Regenaration PGM".Control."metering running" OR
       "Function Ratio check".Control."metering running" OR
       ("Functions"."2k"."pre run program selected" AND "Metering".Metering_running) OR
       "Function Dearing with valve"."Control B"."dearing running") THEN
       "DataloggingDB"."Copy Flush B qty" := true;
   END_IF;

   "R_TRIG_DB_21"(CLK:="DataloggingDB"."Copy Flush B qty" AND NOT ("Function Dearing with valve"."Control B"."dearing running") AND
                  NOT ("Function Regenaration PGM".Control."metering running") AND NOT ("Function Ratio check".Control."metering running") AND
                  NOT ("Functions"."2k"."pre run program selected") AND NOT ("Function Flush"."Control B"."flush running"),
                  Q=>"Temp".bit3);

   IF "R_TRIG_DB_21".Q THEN
       "DataloggingDB".Data_1."Total B flush" := "Flowrate"."Volume in L".mixed + "DataloggingDB".Data_1."Total B flush";
       "DataloggingDB"."Copy Flush B qty" := false;
   END_IF;
END_REGION

REGION Network 5: total Size A
   RUNG wire#powerrail
      Contact( "Metering".Metering_running )
      I_Contact( "Functions"."2k"."pre run program selected" )
      Contact( "Metering".output."ON_outlet Valve A" )
      Coil( "DataloggingDB"."Total Size A calculation"."dosing running" )
   END_RUNG
   RUNG wire#powerrail
      Contact( "DataloggingDB"."Total Size A calculation"."dosing running" )
      Move(in := "Flowrate"."Volume in L"."A", out1 => "DataloggingDB"."Total Size A calculation"."volume dispensed")
   END_RUNG
   RUNG wire#powerrail
      I_Contact( "DataloggingDB"."Total Size A calculation"."dosing running" )
      { S7_Templates := "time_type := Time" } "IEC_Timer_0_DB_81".TON(pt := T#1s, et =>)
      Move(in := 0.0, out1 => "DataloggingDB"."Total Size A calculation"."volume dispensed")
   END_RUNG
   RUNG wire#powerrail
      Contact( "DataloggingDB"."Total Size A calculation"."dosing running" )
      P_Contact(operand := "DataloggingDB"."Ready to Log", bit := "Temp".bit6)
      wire#w1
      { S7_Templates := "SrcType := Real" } Add(in1 := "DataloggingDB"."Total Size A calculation"."volume dispensed", in2 := "DataloggingDB".Data_1."Total size A", out => "DataloggingDB".Data_1."Total size A")
   END_RUNG
   RUNG wire#powerrail
      N_Contact(operand := "DataloggingDB"."Total Size A calculation"."dosing running", bit := "Temp".bit26)
   END_RUNG wire#w1
   // the same network as SCL:
   "DataloggingDB"."Total Size A calculation"."dosing running" := "Metering".Metering_running AND NOT "Functions"."2k"."pre run program selected" AND "Metering".output."ON_outlet Valve A";
   IF "DataloggingDB"."Total Size A calculation"."dosing running" THEN
       "DataloggingDB"."Total Size A calculation"."volume dispensed" := "Flowrate"."Volume in L"."A";
   END_IF;
   "IEC_Timer_0_DB_81".TON(IN := NOT "DataloggingDB"."Total Size A calculation"."dosing running", PT := T#1s);
   IF "IEC_Timer_0_DB_81".Q THEN
       "DataloggingDB"."Total Size A calculation"."volume dispensed" := 0.0;
   END_IF;
   #_w1 := "DataloggingDB"."Total Size A calculation"."dosing running" AND "DataloggingDB"."Ready to Log" AND NOT "Temp".bit6;   // rising edge of "DataloggingDB"."Ready to Log"
   "Temp".bit6 := "DataloggingDB"."Ready to Log";
   #_w2 := NOT "DataloggingDB"."Total Size A calculation"."dosing running" AND "Temp".bit26;   // falling edge of "DataloggingDB"."Total Size A calculation"."dosing running"
   "Temp".bit26 := "DataloggingDB"."Total Size A calculation"."dosing running";
   IF #_w1 OR #_w2 THEN
       "DataloggingDB".Data_1."Total size A" := "DataloggingDB"."Total Size A calculation"."volume dispensed" + "DataloggingDB".Data_1."Total size A";
   END_IF;
END_REGION

REGION Network 6: total Size B
   RUNG wire#powerrail
      Contact( "Metering".Metering_running )
      I_Contact( "Functions"."2k"."pre run program selected" )
      Contact( "Metering".output."ON_outlet valve B" )
      Coil( "DataloggingDB"."Total Size B calculation"."dosing running" )
   END_RUNG
   RUNG wire#powerrail
      Contact( "DataloggingDB"."Total Size B calculation"."dosing running" )
      Move(in := "Flowrate"."Volume in L"."B", out1 => "DataloggingDB"."Total Size B calculation"."volume dispensed")
   END_RUNG
   RUNG wire#powerrail
      I_Contact( "DataloggingDB"."Total Size B calculation"."dosing running" )
      { S7_Templates := "time_type := Time" } "IEC_Timer_0_DB_111".TON(pt := T#1s, et =>)
      Move(in := 0.0, out1 => "DataloggingDB"."Total Size B calculation"."volume dispensed")
   END_RUNG
   RUNG wire#powerrail
      Contact( "DataloggingDB"."Total Size B calculation"."dosing running" )
      P_Contact(operand := "DataloggingDB"."Ready to Log", bit := "Temp".bit9)
      wire#w1
      { S7_Templates := "SrcType := Real" } Add(in1 := "DataloggingDB"."Total Size B calculation"."volume dispensed", in2 := "DataloggingDB".Data_1."Total size B", out => "DataloggingDB".Data_1."Total size B")
   END_RUNG
   RUNG wire#powerrail
      N_Contact(operand := "DataloggingDB"."Total Size B calculation"."dosing running", bit := "Temp".bit19)
   END_RUNG wire#w1
   // the same network as SCL:
   "DataloggingDB"."Total Size B calculation"."dosing running" := "Metering".Metering_running AND NOT "Functions"."2k"."pre run program selected" AND "Metering".output."ON_outlet valve B";
   IF "DataloggingDB"."Total Size B calculation"."dosing running" THEN
       "DataloggingDB"."Total Size B calculation"."volume dispensed" := "Flowrate"."Volume in L"."B";
   END_IF;
   "IEC_Timer_0_DB_111".TON(IN := NOT "DataloggingDB"."Total Size B calculation"."dosing running", PT := T#1s);
   IF "IEC_Timer_0_DB_111".Q THEN
       "DataloggingDB"."Total Size B calculation"."volume dispensed" := 0.0;
   END_IF;
   #_w1 := "DataloggingDB"."Total Size B calculation"."dosing running" AND "DataloggingDB"."Ready to Log" AND NOT "Temp".bit9;   // rising edge of "DataloggingDB"."Ready to Log"
   "Temp".bit9 := "DataloggingDB"."Ready to Log";
   #_w2 := NOT "DataloggingDB"."Total Size B calculation"."dosing running" AND "Temp".bit19;   // falling edge of "DataloggingDB"."Total Size B calculation"."dosing running"
   "Temp".bit19 := "DataloggingDB"."Total Size B calculation"."dosing running";
   IF #_w1 OR #_w2 THEN
       "DataloggingDB".Data_1."Total size B" := "DataloggingDB"."Total Size B calculation"."volume dispensed" + "DataloggingDB".Data_1."Total size B";
   END_IF;
END_REGION

REGION Network 7: Total size
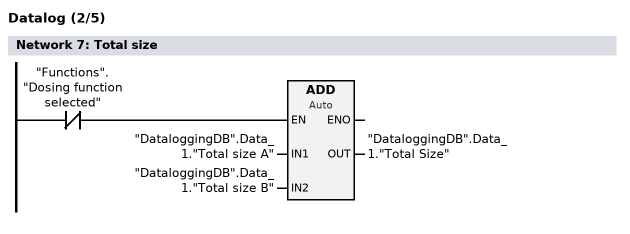
   RUNG wire#powerrail
      I_Contact( "Functions"."Dosing function selected" )
      Add(in1 := "DataloggingDB".Data_1."Total size A", in2 := "DataloggingDB".Data_1."Total size B", out => "DataloggingDB".Data_1."Total Size")
   END_RUNG
   // the same network as SCL:
   IF NOT "Functions"."Dosing function selected" THEN
       "DataloggingDB".Data_1."Total Size" := "DataloggingDB".Data_1."Total size A" + "DataloggingDB".Data_1."Total size B";
   END_IF;
END_REGION

REGION Network 8: Metering Size
END_REGION

REGION Network 9: Shot Size A
END_REGION

REGION Network 10: Shot Size B
END_REGION

REGION Network 11: Mixing Ratio
END_REGION

REGION Network 12: ratio Min
END_REGION

REGION Network 13: ratio Max
END_REGION

REGION Network 14: Volume_Dispensed
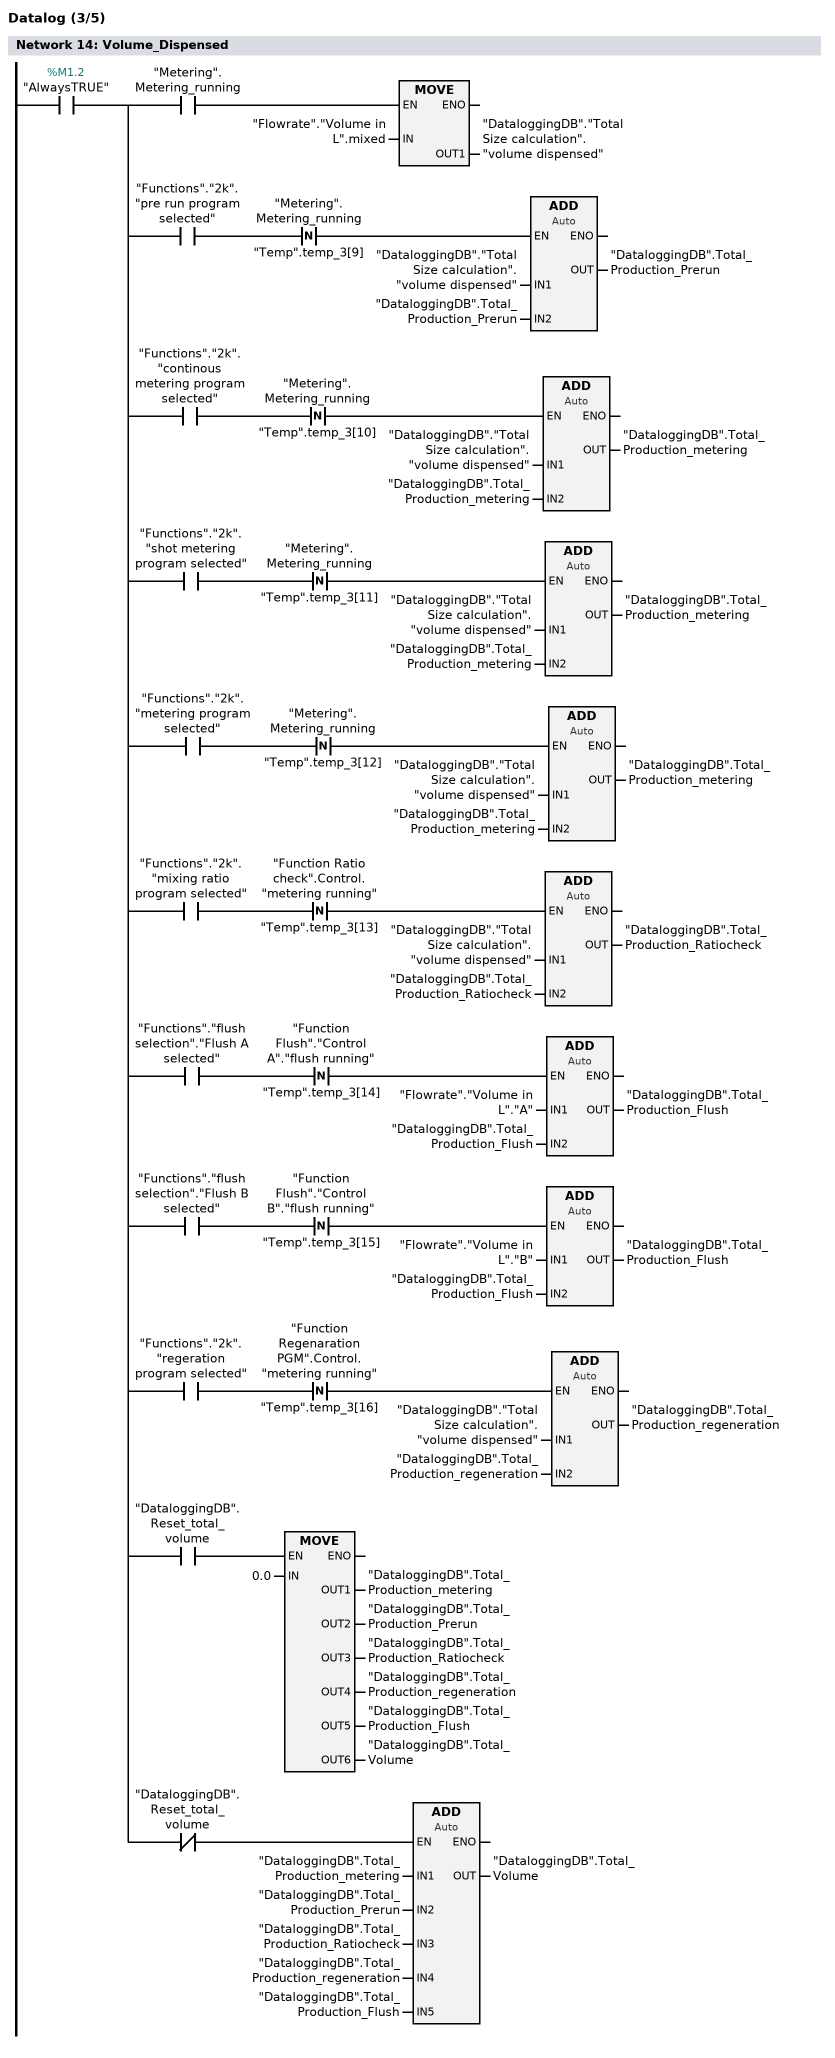
   RUNG wire#powerrail
      Contact( "AlwaysTRUE" )
      wire#w1
      Contact( "Metering".Metering_running )
      Move(in := "Flowrate"."Volume in L".mixed, out1 => "DataloggingDB"."Total Size calculation"."volume dispensed")
   END_RUNG
   RUNG wire#w1
      Contact( "Functions"."2k"."pre run program selected" )
      N_Contact(operand := "Metering".Metering_running, bit := "Temp".temp_3[9])
      Add(in1 := "DataloggingDB"."Total Size calculation"."volume dispensed", in2 := "DataloggingDB".Total_Production_Prerun, out => "DataloggingDB".Total_Production_Prerun)
   END_RUNG
   RUNG wire#w1
      Contact( "Functions"."2k"."continous metering program selected" )
      N_Contact(operand := "Metering".Metering_running, bit := "Temp".temp_3[10])
      Add(in1 := "DataloggingDB"."Total Size calculation"."volume dispensed", in2 := "DataloggingDB".Total_Production_metering, out => "DataloggingDB".Total_Production_metering)
   END_RUNG
   RUNG wire#w1
      Contact( "Functions"."2k"."shot metering program selected" )
      N_Contact(operand := "Metering".Metering_running, bit := "Temp".temp_3[11])
      Add(in1 := "DataloggingDB"."Total Size calculation"."volume dispensed", in2 := "DataloggingDB".Total_Production_metering, out => "DataloggingDB".Total_Production_metering)
   END_RUNG
   RUNG wire#w1
      Contact( "Functions"."2k"."metering program selected" )
      N_Contact(operand := "Metering".Metering_running, bit := "Temp".temp_3[12])
      Add(in1 := "DataloggingDB"."Total Size calculation"."volume dispensed", in2 := "DataloggingDB".Total_Production_metering, out => "DataloggingDB".Total_Production_metering)
   END_RUNG
   RUNG wire#w1
      Contact( "Functions"."2k"."mixing ratio program selected" )
      N_Contact(operand := "Function Ratio check".Control."metering running", bit := "Temp".temp_3[13])
      Add(in1 := "DataloggingDB"."Total Size calculation"."volume dispensed", in2 := "DataloggingDB".Total_Production_Ratiocheck, out => "DataloggingDB".Total_Production_Ratiocheck)
   END_RUNG
   RUNG wire#w1
      Contact( "Functions"."flush selection"."Flush A selected" )
      N_Contact(operand := "Function Flush"."Control A"."flush running", bit := "Temp".temp_3[14])
      Add(in1 := "Flowrate"."Volume in L"."A", in2 := "DataloggingDB".Total_Production_Flush, out => "DataloggingDB".Total_Production_Flush)
   END_RUNG
   RUNG wire#w1
      Contact( "Functions"."flush selection"."Flush B selected" )
      N_Contact(operand := "Function Flush"."Control B"."flush running", bit := "Temp".temp_3[15])
      Add(in1 := "Flowrate"."Volume in L"."B", in2 := "DataloggingDB".Total_Production_Flush, out => "DataloggingDB".Total_Production_Flush)
   END_RUNG
   RUNG wire#w1
      Contact( "Functions"."2k"."regeration program selected" )
      N_Contact(operand := "Function Regenaration PGM".Control."metering running", bit := "Temp".temp_3[16])
      Add(in1 := "DataloggingDB"."Total Size calculation"."volume dispensed", in2 := "DataloggingDB".Total_Production_regeneration, out => "DataloggingDB".Total_Production_regeneration)
   END_RUNG
   RUNG wire#w1
      Contact( "DataloggingDB".Reset_total_volume )
      Move(in := 0.0, out1 => "DataloggingDB".Total_Production_metering, out2 => "DataloggingDB".Total_Production_Prerun, out3 => "DataloggingDB".Total_Production_Ratiocheck, out4 => "DataloggingDB".Total_Production_regeneration, out5 => "DataloggingDB".Total_Production_Flush, out6 => "DataloggingDB".Total_Volume)
   END_RUNG
   RUNG wire#w1
      I_Contact( "DataloggingDB".Reset_total_volume )
      Add(in1 := "DataloggingDB".Total_Production_metering, in2 := "DataloggingDB".Total_Production_Prerun, in3 := "DataloggingDB".Total_Production_Ratiocheck, in4 := "DataloggingDB".Total_Production_regeneration, in5 := "DataloggingDB".Total_Production_Flush, out => "DataloggingDB".Total_Volume)
   END_RUNG
   // the same network as SCL:
   IF "AlwaysTRUE" AND "Metering".Metering_running THEN
       "DataloggingDB"."Total Size calculation"."volume dispensed" := "Flowrate"."Volume in L".mixed;
   END_IF;
   #_w1 := "AlwaysTRUE" AND "Functions"."2k"."pre run program selected" AND NOT "Metering".Metering_running AND "Temp".temp_3[9];   // falling edge of "Metering".Metering_running
   "Temp".temp_3[9] := "Metering".Metering_running;
   IF #_w1 THEN
       "DataloggingDB".Total_Production_Prerun := "DataloggingDB"."Total Size calculation"."volume dispensed" + "DataloggingDB".Total_Production_Prerun;
   END_IF;
   #_w2 := "AlwaysTRUE" AND "Functions"."2k"."continous metering program selected" AND NOT "Metering".Metering_running AND "Temp".temp_3[10];   // falling edge of "Metering".Metering_running
   "Temp".temp_3[10] := "Metering".Metering_running;
   IF #_w2 THEN
       "DataloggingDB".Total_Production_metering := "DataloggingDB"."Total Size calculation"."volume dispensed" + "DataloggingDB".Total_Production_metering;
   END_IF;
   #_w3 := "AlwaysTRUE" AND "Functions"."2k"."shot metering program selected" AND NOT "Metering".Metering_running AND "Temp".temp_3[11];   // falling edge of "Metering".Metering_running
   "Temp".temp_3[11] := "Metering".Metering_running;
   IF #_w3 THEN
       "DataloggingDB".Total_Production_metering := "DataloggingDB"."Total Size calculation"."volume dispensed" + "DataloggingDB".Total_Production_metering;
   END_IF;
   #_w4 := "AlwaysTRUE" AND "Functions"."2k"."metering program selected" AND NOT "Metering".Metering_running AND "Temp".temp_3[12];   // falling edge of "Metering".Metering_running
   "Temp".temp_3[12] := "Metering".Metering_running;
   IF #_w4 THEN
       "DataloggingDB".Total_Production_metering := "DataloggingDB"."Total Size calculation"."volume dispensed" + "DataloggingDB".Total_Production_metering;
   END_IF;
   #_w5 := "AlwaysTRUE" AND "Functions"."2k"."mixing ratio program selected" AND NOT "Function Ratio check".Control."metering running" AND "Temp".temp_3[13];   // falling edge of "Function Ratio check".Control."metering running"
   "Temp".temp_3[13] := "Function Ratio check".Control."metering running";
   IF #_w5 THEN
       "DataloggingDB".Total_Production_Ratiocheck := "DataloggingDB"."Total Size calculation"."volume dispensed" + "DataloggingDB".Total_Production_Ratiocheck;
   END_IF;
   #_w6 := "AlwaysTRUE" AND "Functions"."flush selection"."Flush A selected" AND NOT "Function Flush"."Control A"."flush running" AND "Temp".temp_3[14];   // falling edge of "Function Flush"."Control A"."flush running"
   "Temp".temp_3[14] := "Function Flush"."Control A"."flush running";
   IF #_w6 THEN
       "DataloggingDB".Total_Production_Flush := "Flowrate"."Volume in L"."A" + "DataloggingDB".Total_Production_Flush;
   END_IF;
   #_w7 := "AlwaysTRUE" AND "Functions"."flush selection"."Flush B selected" AND NOT "Function Flush"."Control B"."flush running" AND "Temp".temp_3[15];   // falling edge of "Function Flush"."Control B"."flush running"
   "Temp".temp_3[15] := "Function Flush"."Control B"."flush running";
   IF #_w7 THEN
       "DataloggingDB".Total_Production_Flush := "Flowrate"."Volume in L"."B" + "DataloggingDB".Total_Production_Flush;
   END_IF;
   #_w8 := "AlwaysTRUE" AND "Functions"."2k"."regeration program selected" AND NOT "Function Regenaration PGM".Control."metering running" AND "Temp".temp_3[16];   // falling edge of "Function Regenaration PGM".Control."metering running"
   "Temp".temp_3[16] := "Function Regenaration PGM".Control."metering running";
   IF #_w8 THEN
       "DataloggingDB".Total_Production_regeneration := "DataloggingDB"."Total Size calculation"."volume dispensed" + "DataloggingDB".Total_Production_regeneration;
   END_IF;
   IF "AlwaysTRUE" AND "DataloggingDB".Reset_total_volume THEN
       "DataloggingDB".Total_Production_metering := 0.0;
       "DataloggingDB".Total_Production_Prerun := 0.0;
       "DataloggingDB".Total_Production_Ratiocheck := 0.0;
       "DataloggingDB".Total_Production_regeneration := 0.0;
       "DataloggingDB".Total_Production_Flush := 0.0;
       "DataloggingDB".Total_Volume := 0.0;
   END_IF;
   IF "AlwaysTRUE" AND NOT "DataloggingDB".Reset_total_volume THEN
       "DataloggingDB".Total_Volume := "DataloggingDB".Total_Production_metering + "DataloggingDB".Total_Production_Prerun + "DataloggingDB".Total_Production_Ratiocheck + "DataloggingDB".Total_Production_regeneration + "DataloggingDB".Total_Production_Flush;
   END_IF;
END_REGION

REGION Network 15 (SCL)
   IF NOT ("Functions"."Dosing Running") THEN
       "event For datalogging"."event number" := 1; //Event machine idle
   ELSIF "Functions"."2k"."metering program selected" AND "Metering".Metering_running THEN
       "event For datalogging"."event number" := 2; //Event metering program running
   ELSIF "Function Ratio check".Control."metering running" THEN
       "event For datalogging"."event number" := 3; //Event Ratio check program running
   ELSIF "Functions"."2k"."shot metering program selected" AND "Metering".Metering_running THEN
       "event For datalogging"."event number" := 4; //Event metering shot running
   ELSIF "Functions"."2k"."continous metering program selected" AND "Metering".Metering_running THEN
       "event For datalogging"."event number" := 5; //Event metering Continuous metering running
   ELSIF "Functions"."2k"."pre run program selected" AND "Metering".Metering_running THEN
       "event For datalogging"."event number" := 6; //Event "Metering" Pre run running
   ELSIF "Function Flush"."Control A"."flush running" THEN
       "event For datalogging"."event number" := 7; // Event metering Flush running
   ELSIF "Function Dearing with valve"."Control A"."dearing running" OR "Function Dearing with valve"."Control B"."dearing running" THEN
       "event For datalogging"."event number" := 8; // Event deaerate running
   ELSIF "Faults&warnings"."Critical Alarm metering A&B" THEN
       "event For datalogging"."event number" := 9; // Event Machine fault
   ELSIF "Function Regenaration PGM".Control."metering running" THEN
       "event For datalogging"."event number" := 11; // Event regeneration running
   ELSIF "metering Completed" THEN
       "event For datalogging"."event number" := 12; // dosing completed
   END_IF;

   "DataloggingDB".Data.Function := "event For datalogging".Function_String["event For datalogging"."event number"];
END_REGION

REGION Network 16: Function
